LIN {X 0,Y 484.481,Z 413.449,A -85,B 0,C 180,E1 -6825.401,E2 -6825.401} C_VEL
LIN {X 0,Y 484,Z 426.052,A -85,B 0,C 180,E1 -6826.351,E2 -6826.351} C_VEL
LIN {X 0,Y 483.451,Z 437.461,A -85,B 0,C 180,E1 -6827.405,E2 -6827.405} C_VEL
LIN {X 0,Y 482.946,Z 446.93,A -85,B 0,C 180,E1 -6828.457,E2 -6828.457} C_VEL
LIN {X 0,Y 482.492,Z 456.426,A -85,B 0,C 180,E1 -6829.721,E2 -6829.721} C_VEL
LIN {X 0,Y 482.084,Z 465.497,A -85,B 0,C 180,E1 -6831.195,E2 -6831.195} C_VEL
LIN {X 0,Y 481.802,Z 471.841,A -85,B 0,C 180,E1 -6832.456,E2 -6832.456} C_VEL
LIN {X 0,Y 481.631,Z 477.067,A -85,B 0,C 180,E1 -6833.717,E2 -6833.717} C_VEL
LIN {X 0,Y 481.446,Z 482.599,A -85,B 0,C 180,E1 -6835.395,E2 -6835.395} C_VEL
LIN {X 0,Y 481.292,Z 485.698,A -85,B 0,C 180,E1 -6836.651,E2 -6836.651} C_VEL
LIN {X 0,Y 481.216,Z 488.621,A -85,B 0,C 180,E1 -6838.326,E2 -6838.326} C_VEL
LIN {X 0,Y 481.127,Z 490.218,A -85,B 0,C 180,E1 -6840,E2 -6840} C_VEL
LIN {X 0,Y 481.209,Z 490.492,A -85,B 0,C 180,E1 -6841.674,E2 -6841.674} C_VEL
LIN {X 0,Y 481.255,Z 489.477,A -85,B 0,C 180,E1 -6843.349,E2 -6843.349} C_VEL
LIN {X 0,Y 481.353,Z 487.122,A -85,B 0,C 180,E1 -6845.026,E2 -6845.026} C_VEL
LIN {X 0,Y 481.497,Z 484.405,A -85,B 0,C 180,E1 -6846.285,E2 -6846.285} C_VEL
LIN {X 0,Y 481.752,Z 479.514,A -85,B 0,C 180,E1 -6847.966,E2 -6847.966} C_VEL
LIN {X 0,Y 481.884,Z 474.735,A -85,B 0,C 180,E1 -6849.232,E2 -6849.232} C_VEL
LIN {X 0,Y 482.239,Z 467.834,A -85,B 0,C 180,E1 -6850.708,E2 -6850.708} C_VEL
LIN {X 0,Y 482.693,Z 459.289,A -85,B 0,C 180,E1 -6852.178,E2 -6852.178} C_VEL
LIN {X 0,Y 483.198,Z 450.109,A -85,B 0,C 180,E1 -6853.457,E2 -6853.457} C_VEL
LIN {X 0,Y 483.682,Z 438.95,A -85,B 0,C 180,E1 -6854.731,E2 -6854.731} C_VEL
LIN {X 0,Y 484.26,Z 427.523,A -85,B 0,C 180,E1 -6855.79,E2 -6855.79} C_VEL
LIN {X 0,Y 484.738,Z 415.459,A -85,B 0,C 180,E1 -6856.702,E2 -6856.702} C_VEL
LIN {X 0,Y 485.245,Z 402.361,A -85,B 0,C 180,E1 -6857.489,E2 -6857.489} C_VEL
LIN {X 0,Y 485.233,Z 400.246,A -85,B 0,C 180,E1 -6857.598,E2 -6857.598} C_VEL
LIN {X 0,Y 481.758,Z 389.103,A -85,B 0,C 180,E1 -6858.288,E2 -6858.288} C_VEL
LIN {X 0,Y 481.651,Z 389.119,A -85,B 0,C 180,E1 -6861.394,E2 -6861.394} C_VEL
LIN {X 0,Y 481.681,Z 389.115,A -85,B 0,C 180,E1 -6864.113,E2 -6864.113} C_VEL
LIN {X 0,Y 481.75,Z 389.103,A -85,B 0,C 180,E1 -6867.139,E2 -6867.139} C_VEL
LIN {X 0,Y 481.682,Z 389.111,A -85,B 0,C 180,E1 -6869.741,E2 -6869.741} C_VEL
LIN {X 0,Y 481.675,Z 389.113,A -85,B 0,C 180,E1 -6872.674,E2 -6872.674} C_VEL
LIN {X 0,Y 481.639,Z 389.117,A -85,B 0,C 180,E1 -6875.709,E2 -6875.709} C_VEL
LIN {X 0,Y 481.673,Z 389.114,A -85,B 0,C 180,E1 -6878.859,E2 -6878.859} C_VEL
LIN {X 0,Y 481.656,Z 389.115,A -85,B 0,C 180,E1 -6881.913,E2 -6881.913} C_VEL
LIN {X 0,Y 481.663,Z 389.116,A -85,B 0,C 180,E1 -6884.457,E2 -6884.457} C_VEL
LIN {X 0,Y 481.651,Z 389.119,A -85,B 0,C 180,E1 -6887.839,E2 -6887.839} C_VEL
LIN {X 0,Y 481.704,Z 389.203,A -85,B 0,C 180,E1 -6888.406,E2 -6888.406} C_VEL
LIN {X 0,Y 483.139,Z 396.916,A -85,B 0,C 180,E1 -6890.887,E2 -6890.887} C_VEL
LIN {X 0,Y 483.245,Z 401.045,A -85,B 0,C 180,E1 -6892.046,E2 -6892.046} C_VEL
LIN {X 0,Y 482.441,Z 414.228,A -85,B 0,C 180,E1 -6895.379,E2 -6895.379} C_VEL
LIN {X 0,Y 482.294,Z 426.909,A -85,B 0,C 180,E1 -6898.358,E2 -6898.358} C_VEL
LIN {X 0,Y 482.22,Z 439.845,A -85,B 0,C 180,E1 -6901.252,E2 -6901.252} C_VEL
LIN {X 0,Y 482.05,Z 455.738,A -85,B 0,C 180,E1 -6904.679,E2 -6904.679} C_VEL
LIN {X 0,Y 481.88,Z 471.239,A -85,B 0,C 180,E1 -6907.941,E2 -6907.941} C_VEL
LIN {X 0,Y 481.707,Z 486.219,A -85,B 0,C 180,E1 -6911.057,E2 -6911.057} C_VEL
LIN {X 0,Y 481.693,Z 490.574,A -85,B 0,C 180,E1 -6911.957,E2 -6911.957} C_VEL
LIN {X 0,Y 483.326,Z 507.533,A -85,B 0,C 180,E1 -6912.397,E2 -6912.397} C_VEL
LIN {X 0,Y 484.795,Z 517.449,A -85,B 0,C 180,E1 -6912.765,E2 -6912.765} C_VEL
LIN {X 0,Y 484.293,Z 531.486,A -85,B 0,C 180,E1 -6913.342,E2 -6913.342} C_VEL
LIN {X 0,Y 483.695,Z 545.297,A -85,B 0,C 180,E1 -6914.082,E2 -6914.082} C_VEL
LIN {X 0,Y 483.143,Z 559.303,A -85,B 0,C 180,E1 -6915.036,E2 -6915.036} C_VEL
LIN {X 0,Y 482.585,Z 571.818,A -85,B 0,C 180,E1 -6916.095,E2 -6916.095} C_VEL
LIN {X 0,Y 482.176,Z 582.238,A -85,B 0,C 180,E1 -6917.156,E2 -6917.156} C_VEL
LIN {X 0,Y 481.863,Z 592.671,A -85,B 0,C 180,E1 -6918.43,E2 -6918.43} C_VEL
LIN {X 0,Y 481.477,Z 601.314,A -85,B 0,C 180,E1 -6919.699,E2 -6919.699} C_VEL
LIN {X 0,Y 481.308,Z 609.635,A -85,B 0,C 180,E1 -6921.18,E2 -6921.18} C_VEL
LIN {X 0,Y 481.142,Z 615.438,A -85,B 0,C 180,E1 -6922.445,E2 -6922.445} C_VEL
LIN {X 0,Y 481.117,Z 620.135,A -85,B 0,C 180,E1 -6923.675,E2 -6923.675} C_VEL
LIN {X 0,Y 481.094,Z 624.005,A -85,B 0,C 180,E1 -6924.971,E2 -6924.971} C_VEL
LIN {X 0,Y 481.1,Z 626.043,A -85,B 0,C 180,E1 -6925.81,E2 -6925.81} C_VEL
LIN {X 0,Y 481.01,Z 628.967,A -85,B 0,C 180,E1 -6927.487,E2 -6927.487} C_VEL
LIN {X 0,Y 480.936,Z 630.44,A -85,B 0,C 180,E1 -6929.162,E2 -6929.162} C_VEL
LIN {X 0,Y 480.995,Z 630.658,A -85,B 0,C 180,E1 -6929.999,E2 -6929.999} C_VEL
LIN {X 0,Y 480.955,Z 630.008,A -85,B 0,C 180,E1 -6931.674,E2 -6931.674} C_VEL
LIN {X 0,Y 481.003,Z 627.954,A -85,B 0,C 180,E1 -6933.35,E2 -6933.35} C_VEL
LIN {X 0,Y 481.054,Z 624.44,A -85,B 0,C 180,E1 -6935.028,E2 -6935.028} C_VEL
LIN {X 0,Y 481.076,Z 619.364,A -85,B 0,C 180,E1 -6936.711,E2 -6936.711} C_VEL
LIN {X 0,Y 481.208,Z 612.595,A -85,B 0,C 180,E1 -6938.397,E2 -6938.397} C_VEL
LIN {X 0,Y 481.392,Z 605.054,A -85,B 0,C 180,E1 -6939.876,E2 -6939.876} C_VEL
LIN {X 0,Y 481.762,Z 595.692,A -85,B 0,C 180,E1 -6941.357,E2 -6941.357} C_VEL
LIN {X 0,Y 482.122,Z 585.91,A -85,B 0,C 180,E1 -6942.629,E2 -6942.629} C_VEL
LIN {X 0,Y 482.589,Z 575.113,A -85,B 0,C 180,E1 -6943.795,E2 -6943.795} C_VEL
LIN {X 0,Y 483.117,Z 563.234,A -85,B 0,C 180,E1 -6944.855,E2 -6944.855} C_VEL
LIN {X 0,Y 483.718,Z 551.697,A -85,B 0,C 180,E1 -6945.699,E2 -6945.699} C_VEL
LIN {X 0,Y 484.311,Z 539,A -85,B 0,C 180,E1 -6946.453,E2 -6946.453} C_VEL
LIN {X 0,Y 484.793,Z 525.706,A -85,B 0,C 180,E1 -6947.07,E2 -6947.07} C_VEL
LIN {X 0,Y 484.895,Z 515.976,A -85,B 0,C 180,E1 -6947.427,E2 -6947.427} C_VEL
LIN {X 0,Y 483.035,Z 503.611,A -85,B 0,C 180,E1 -6947.833,E2 -6947.833} C_VEL
LIN {X 0,Y 481.739,Z 494.305,A -85,B 0,C 180,E1 -6948.071,E2 -6948.071} C_VEL
LIN {X 0,Y 482.024,Z 480.891,A -85,B 0,C 180,E1 -6951.072,E2 -6951.072} C_VEL
LIN {X 0,Y 482.329,Z 469.472,A -85,B 0,C 180,E1 -6953.674,E2 -6953.674} C_VEL
LIN {X 0,Y 482.755,Z 455.849,A -85,B 0,C 180,E1 -6956.826,E2 -6956.826} C_VEL
LIN {X 0,Y 483.3,Z 442.011,A -85,B 0,C 180,E1 -6960.11,E2 -6960.11} C_VEL
LIN {X 0,Y 483.812,Z 428.138,A -85,B 0,C 180,E1 -6963.503,E2 -6963.503} C_VEL
LIN {X 0,Y 484.574,Z 413.921,A -85,B 0,C 180,E1 -6967.09,E2 -6967.09} C_VEL
LIN {X 0,Y 484.908,Z 406.263,A -85,B 0,C 180,E1 -6969.083,E2 -6969.083} C_VEL
LIN {X 0,Y 484.024,Z 400.159,A -85,B 0,C 180,E1 -6970.796,E2 -6970.796} C_VEL
LIN {X 0,Y 481.859,Z 390.061,A -85,B 0,C 180,E1 -6973.787,E2 -6973.787} C_VEL
LIN {X 0,Y 481.67,Z 389.114,A -85,B 0,C 180,E1 -6974.107,E2 -6974.107} C_VEL
LIN {X 0,Y 481.682,Z 389.107,A -85,B 0,C 180,E1 -6976.845,E2 -6976.845} C_VEL
LIN {X 0,Y 481.705,Z 389.108,A -85,B 0,C 180,E1 -6980.062,E2 -6980.062} C_VEL
LIN {X 0,Y 481.624,Z 389.118,A -85,B 0,C 180,E1 -6983.374,E2 -6983.374} C_VEL
LIN {X 0,Y 481.7,Z 389.106,A -85,B 0,C 180,E1 -6986.329,E2 -6986.329} C_VEL
LIN {X 0,Y 481.649,Z 389.116,A -85,B 0,C 180,E1 -6989.415,E2 -6989.415} C_VEL
LIN {X 0,Y 481.693,Z 389.108,A -85,B 0,C 180,E1 -6992.168,E2 -6992.168} C_VEL
LIN {X 0,Y 481.708,Z 389.105,A -85,B 0,C 180,E1 -6994.969,E2 -6994.969} C_VEL
LIN {X 0,Y 481.64,Z 389.115,A -85,B 0,C 180,E1 -6997.704,E2 -6997.704} C_VEL
LIN {X 0,Y 481.697,Z 389.106,A -85,B 0,C 180,E1 -7000.393,E2 -7000.393} C_VEL
LIN {X 0,Y 481.682,Z 389.109,A -85,B 0,C 180,E1 -7003.034,E2 -7003.034} C_VEL
LIN {X 0,Y 481.683,Z 389.11,A -85,B 0,C 180,E1 -7005.639,E2 -7005.639} C_VEL
LIN {X 0,Y 481.784,Z 389.096,A -85,B 0,C 180,E1 -7008.216,E2 -7008.216} C_VEL
LIN {X 0,Y 481.753,Z 389.101,A -85,B 0,C 180,E1 -7011.612,E2 -7011.612} C_VEL
LIN {X 0,Y 481.807,Z 389.093,A -85,B 0,C 180,E1 -7014.14,E2 -7014.14} C_VEL
LIN {X 0,Y 481.919,Z 389.081,A -85,B 0,C 180,E1 -7017.493,E2 -7017.493} C_VEL
LIN {X 0,Y 481.93,Z 389.078,A -85,B 0,C 180,E1 -7020,E2 -7020} C_VEL
LIN {X 0,Y 481.919,Z 389.078,A -85,B 0,C 180,E1 -7022.508,E2 -7022.508} C_VEL
LIN {X 0,Y 481.812,Z 389.093,A -85,B 0,C 180,E1 -7025.861,E2 -7025.861} C_VEL
LIN {X 0,Y 481.754,Z 389.099,A -85,B 0,C 180,E1 -7028.389,E2 -7028.389} C_VEL
LIN {X 0,Y 481.786,Z 389.096,A -85,B 0,C 180,E1 -7031.784,E2 -7031.784} C_VEL
LIN {X 0,Y 481.732,Z 389.105,A -85,B 0,C 180,E1 -7035.225,E2 -7035.225} C_VEL
LIN {X 0,Y 481.703,Z 389.106,A -85,B 0,C 180,E1 -7038.722,E2 -7038.722} C_VEL
LIN {X 0,Y 481.637,Z 389.116,A -85,B 0,C 180,E1 -7041.395,E2 -7041.395} C_VEL
LIN {X 0,Y 481.668,Z 389.11,A -85,B 0,C 180,E1 -7044.114,E2 -7044.114} C_VEL
LIN {X 0,Y 481.744,Z 389.104,A -85,B 0,C 180,E1 -7047.141,E2 -7047.141} C_VEL
LIN {X 0,Y 481.671,Z 389.111,A -85,B 0,C 180,E1 -7049.742,E2 -7049.742} C_VEL
LIN {X 0,Y 481.666,Z 389.111,A -85,B 0,C 180,E1 -7052.675,E2 -7052.675} C_VEL
LIN {X 0,Y 481.636,Z 389.115,A -85,B 0,C 180,E1 -7055.71,E2 -7055.71} C_VEL
LIN {X 0,Y 481.665,Z 389.114,A -85,B 0,C 180,E1 -7058.86,E2 -7058.86} C_VEL
LIN {X 0,Y 481.657,Z 389.111,A -85,B 0,C 180,E1 -7061.915,E2 -7061.915} C_VEL
LIN {X 0,Y 481.655,Z 389.112,A -85,B 0,C 180,E1 -7064.458,E2 -7064.458} C_VEL
LIN {X 0,Y 481.645,Z 389.113,A -85,B 0,C 180,E1 -7067.841,E2 -7067.841} C_VEL
LIN {X 0,Y 481.716,Z 389.106,A -85,B 0,C 180,E1 -7070.647,E2 -7070.647} C_VEL
LIN {X 0,Y 481.641,Z 389.113,A -85,B 0,C 180,E1 -7074.292,E2 -7074.292} C_VEL
LIN {X 0,Y 481.672,Z 389.111,A -85,B 0,C 180,E1 -7077.327,E2 -7077.327} C_VEL
LIN {X 0,Y 481.678,Z 389.109,A -85,B 0,C 180,E1 -7080.26,E2 -7080.26} C_VEL
LIN {X 0,Y 481.745,Z 389.102,A -85,B 0,C 180,E1 -7083.113,E2 -7083.113} C_VEL
LIN {X 0,Y 481.674,Z 389.109,A -85,B 0,C 180,E1 -7085.888,E2 -7085.888} C_VEL
LIN {X 0,Y 481.636,Z 389.113,A -85,B 0,C 180,E1 -7087.993,E2 -7087.993} C_VEL
LIN {X 0,Y 480.97,Z 389.201,A -85,B 0,C 180,E1 -7088.691,E2 -7088.691} C_VEL
LIN {X 0,Y 478.144,Z 389.55,A -85,B 0,C 180,E1 -7089.826,E2 -7089.826} C_VEL
LIN {X 0,Y 475.759,Z 389.85,A -85,B 0,C 180,E1 -7090.74,E2 -7090.74} C_VEL
LIN {X 0,Y 474.738,Z 389.974,A -85,B 0,C 180,E1 -7091.446,E2 -7091.446} C_VEL
LIN {X 0,Y 474.656,Z 389.983,A -85,B 0,C 180,E1 -7091.685,E2 -7091.685} C_VEL
LIN {X 0,Y 474.667,Z 389.985,A -85,B 0,C 180,E1 -7094.544,E2 -7094.544} C_VEL
LIN {X 0,Y 474.411,Z 390.02,A -85,B 0,C 180,E1 -7097.971,E2 -7097.971} C_VEL
LIN {X 0,Y 477.563,Z 400.909,A -85,B 0,C 180,E1 -7098.38,E2 -7098.38} C_VEL
LIN {X 0,Y 477.396,Z 412.945,A -85,B 0,C 180,E1 -7098.86,E2 -7098.86} C_VEL
LIN {X 0,Y 477.088,Z 424.636,A -85,B 0,C 180,E1 -7099.498,E2 -7099.498} C_VEL
LIN {X 0,Y 476.667,Z 436.587,A -85,B 0,C 180,E1 -7100.346,E2 -7100.346} C_VEL
LIN {X 0,Y 476.218,Z 447.382,A -85,B 0,C 180,E1 -7101.322,E2 -7101.322} C_VEL
LIN {X 0,Y 475.777,Z 456.619,A -85,B 0,C 180,E1 -7102.361,E2 -7102.361} C_VEL
LIN {X 0,Y 475.463,Z 465.754,A -85,B 0,C 180,E1 -7103.636,E2 -7103.636} C_VEL
LIN {X 0,Y 475.01,Z 473.056,A -85,B 0,C 180,E1 -7104.908,E2 -7104.908} C_VEL
LIN {X 0,Y 474.819,Z 478.896,A -85,B 0,C 180,E1 -7106.182,E2 -7106.182} C_VEL
LIN {X 0,Y 474.549,Z 483.539,A -85,B 0,C 180,E1 -7107.454,E2 -7107.454} C_VEL
LIN {X 0,Y 474.42,Z 487.086,A -85,B 0,C 180,E1 -7108.728,E2 -7108.728} C_VEL
LIN {X 0,Y 474.264,Z 489.665,A -85,B 0,C 180,E1 -7110.001,E2 -7110.001} C_VEL
LIN {X 0,Y 474.172,Z 490.883,A -85,B 0,C 180,E1 -7110.85,E2 -7110.85} C_VEL
LIN {X 0,Y 474.231,Z 491.699,A -85,B 0,C 180,E1 -7111.699,E2 -7111.699} C_VEL
LIN {X 0,Y 474.199,Z 492.137,A -85,B 0,C 180,E1 -7113.4,E2 -7113.4} C_VEL
LIN {X 0,Y 474.326,Z 491.062,A -85,B 0,C 180,E1 -7115.101,E2 -7115.101} C_VEL
LIN {X 0,Y 474.401,Z 488.37,A -85,B 0,C 180,E1 -7116.807,E2 -7116.807} C_VEL
LIN {X 0,Y 474.51,Z 485.252,A -85,B 0,C 180,E1 -7118.089,E2 -7118.089} C_VEL
LIN {X 0,Y 474.746,Z 481.073,A -85,B 0,C 180,E1 -7119.373,E2 -7119.373} C_VEL
LIN {X 0,Y 475,Z 475.726,A -85,B 0,C 180,E1 -7120.659,E2 -7120.659} C_VEL
LIN {X 0,Y 475.219,Z 469.012,A -85,B 0,C 180,E1 -7121.95,E2 -7121.95} C_VEL
LIN {X 0,Y 475.672,Z 460.54,A -85,B 0,C 180,E1 -7123.24,E2 -7123.24} C_VEL
LIN {X 0,Y 476.07,Z 451.844,A -85,B 0,C 180,E1 -7124.317,E2 -7124.317} C_VEL
LIN {X 0,Y 476.483,Z 442.254,A -85,B 0,C 180,E1 -7125.288,E2 -7125.288} C_VEL
LIN {X 0,Y 476.917,Z 431.6,A -85,B 0,C 180,E1 -7126.15,E2 -7126.15} C_VEL
LIN {X 0,Y 477.284,Z 419.943,A -85,B 0,C 180,E1 -7126.895,E2 -7126.895} C_VEL
LIN {X 0,Y 477.516,Z 408.575,A -85,B 0,C 180,E1 -7127.451,E2 -7127.451} C_VEL
LIN {X 0,Y 477.528,Z 400.444,A -85,B 0,C 180,E1 -7127.755,E2 -7127.755} C_VEL
LIN {X 0,Y 474.357,Z 390.025,A -85,B 0,C 180,E1 -7128.162,E2 -7128.162} C_VEL
LIN {X 0,Y 474.575,Z 389.998,A -85,B 0,C 180,E1 -7131.096,E2 -7131.096} C_VEL
LIN {X 0,Y 474.663,Z 389.982,A -85,B 0,C 180,E1 -7134.493,E2 -7134.493} C_VEL
LIN {X 0,Y 474.687,Z 389.981,A -85,B 0,C 180,E1 -7137.335,E2 -7137.335} C_VEL
LIN {X 0,Y 474.611,Z 389.99,A -85,B 0,C 180,E1 -7140.23,E2 -7140.23} C_VEL
LIN {X 0,Y 474.631,Z 389.989,A -85,B 0,C 180,E1 -7143.222,E2 -7143.222} C_VEL
LIN {X 0,Y 474.594,Z 389.994,A -85,B 0,C 180,E1 -7146.324,E2 -7146.324} C_VEL
LIN {X 0,Y 474.623,Z 389.983,A -85,B 0,C 180,E1 -7149.646,E2 -7149.646} C_VEL
LIN {X 0,Y 474.62,Z 389.988,A -85,B 0,C 180,E1 -7152.934,E2 -7152.934} C_VEL
LIN {X 0,Y 474.621,Z 389.986,A -85,B 0,C 180,E1 -7155.896,E2 -7155.896} C_VEL
LIN {X 0,Y 474.638,Z 389.98,A -85,B 0,C 180,E1 -7159.04,E2 -7159.04} C_VEL
LIN {X 0,Y 474.616,Z 389.973,A -85,B 0,C 180,E1 -7161.704,E2 -7161.704} C_VEL
LIN {X 0,Y 474.634,Z 389.985,A -85,B 0,C 180,E1 -7164.726,E2 -7164.726} C_VEL
LIN {X 0,Y 474.64,Z 389.984,A -85,B 0,C 180,E1 -7167.788,E2 -7167.788} C_VEL
LIN {X 0,Y 474.627,Z 389.966,A -85,B 0,C 180,E1 -7170.885,E2 -7170.885} C_VEL
LIN {X 0,Y 474.658,Z 389.981,A -85,B 0,C 180,E1 -7173.628,E2 -7173.628} C_VEL
LIN {X 0,Y 474.639,Z 389.984,A -85,B 0,C 180,E1 -7176.642,E2 -7176.642} C_VEL
LIN {X 0,Y 474.658,Z 389.983,A -85,B 0,C 180,E1 -7180.089,E2 -7180.089} C_VEL
LIN {X 0,Y 474.643,Z 389.986,A -85,B 0,C 180,E1 -7182.774,E2 -7182.774} C_VEL
LIN {X 0,Y 474.66,Z 389.987,A -85,B 0,C 180,E1 -7183.698,E2 -7183.698} C_VEL
LIN {X 0,Y 478.112,Z 401.182,A -85,B 0,C 180,E1 -7184.391,E2 -7184.391} C_VEL
LIN {X 0,Y 477.676,Z 414.246,A -85,B 0,C 180,E1 -7185.188,E2 -7185.188} C_VEL
LIN {X 0,Y 477.171,Z 426.871,A -85,B 0,C 180,E1 -7186.152,E2 -7186.152} C_VEL
LIN {X 0,Y 476.591,Z 438.305,A -85,B 0,C 180,E1 -7187.22,E2 -7187.22} C_VEL
LIN {X 0,Y 476.047,Z 447.801,A -85,B 0,C 180,E1 -7188.288,E2 -7188.288} C_VEL
LIN {X 0,Y 475.566,Z 457.324,A -85,B 0,C 180,E1 -7189.57,E2 -7189.57} C_VEL
LIN {X 0,Y 475.14,Z 466.422,A -85,B 0,C 180,E1 -7191.065,E2 -7191.065} C_VEL
LIN {X 0,Y 474.77,Z 474.16,A -85,B 0,C 180,E1 -7192.659,E2 -7192.659} C_VEL
LIN {X 0,Y 474.568,Z 479.586,A -85,B 0,C 180,E1 -7194.05,E2 -7194.05} C_VEL
LIN {X 0,Y 474.371,Z 484.706,A -85,B 0,C 180,E1 -7195.752,E2 -7195.752} C_VEL
LIN {X 0,Y 474.191,Z 488.351,A -85,B 0,C 180,E1 -7197.451,E2 -7197.451} C_VEL
LIN {X 0,Y 474.131,Z 490.614,A -85,B 0,C 180,E1 -7199.15,E2 -7199.15} C_VEL
LIN {X 0,Y 474.13,Z 491.557,A -85,B 0,C 180,E1 -7200.849,E2 -7200.849} C_VEL
LIN {X 0,Y 474.188,Z 491.196,A -85,B 0,C 180,E1 -7202.548,E2 -7202.548} C_VEL
LIN {X 0,Y 474.302,Z 489.516,A -85,B 0,C 180,E1 -7204.249,E2 -7204.249} C_VEL
LIN {X 0,Y 474.548,Z 486.437,A -85,B 0,C 180,E1 -7205.95,E2 -7205.95} C_VEL
LIN {X 0,Y 474.668,Z 481.914,A -85,B 0,C 180,E1 -7207.658,E2 -7207.658} C_VEL
LIN {X 0,Y 474.946,Z 475.768,A -85,B 0,C 180,E1 -7209.368,E2 -7209.368} C_VEL
LIN {X 0,Y 475.329,Z 468.849,A -85,B 0,C 180,E1 -7210.866,E2 -7210.866} C_VEL
LIN {X 0,Y 475.825,Z 460.26,A -85,B 0,C 180,E1 -7212.356,E2 -7212.356} C_VEL
LIN {X 0,Y 476.362,Z 451.042,A -85,B 0,C 180,E1 -7213.654,E2 -7213.654} C_VEL
LIN {X 0,Y 476.897,Z 439.881,A -85,B 0,C 180,E1 -7214.945,E2 -7214.945} C_VEL
LIN {X 0,Y 477.509,Z 428.474,A -85,B 0,C 180,E1 -7216.019,E2 -7216.019} C_VEL
LIN {X 0,Y 478.025,Z 416.614,A -85,B 0,C 180,E1 -7216.931,E2 -7216.931} C_VEL
LIN {X 0,Y 478.544,Z 403.318,A -85,B 0,C 180,E1 -7217.742,E2 -7217.742} C_VEL
LIN {X 0,Y 478.234,Z 401.241,A -85,B 0,C 180,E1 -7217.865,E2 -7217.865} C_VEL
LIN {X 0,Y 474.681,Z 389.984,A -85,B 0,C 180,E1 -7218.584,E2 -7218.584} C_VEL
LIN {X 0,Y 474.638,Z 389.99,A -85,B 0,C 180,E1 -7221.116,E2 -7221.116} C_VEL
LIN {X 0,Y 474.662,Z 389.988,A -85,B 0,C 180,E1 -7224.493,E2 -7224.493} C_VEL
LIN {X 0,Y 474.684,Z 389.983,A -85,B 0,C 180,E1 -7227.334,E2 -7227.334} C_VEL
LIN {X 0,Y 474.608,Z 389.992,A -85,B 0,C 180,E1 -7230.23,E2 -7230.23} C_VEL
LIN {X 0,Y 474.646,Z 389.987,A -85,B 0,C 180,E1 -7233.22,E2 -7233.22} C_VEL
LIN {X 0,Y 474.591,Z 389.995,A -85,B 0,C 180,E1 -7236.323,E2 -7236.323} C_VEL
LIN {X 0,Y 474.63,Z 389.99,A -85,B 0,C 180,E1 -7239.647,E2 -7239.647} C_VEL
LIN {X 0,Y 474.618,Z 389.993,A -85,B 0,C 180,E1 -7242.934,E2 -7242.934} C_VEL
LIN {X 0,Y 474.612,Z 389.995,A -85,B 0,C 180,E1 -7245.895,E2 -7245.895} C_VEL
LIN {X 0,Y 474.65,Z 390.163,A -85,B 0,C 180,E1 -7248.052,E2 -7248.052} C_VEL
LIN {X 0,Y 476.134,Z 397.733,A -85,B 0,C 180,E1 -7250.601,E2 -7250.601} C_VEL
LIN {X 0,Y 476.361,Z 401.493,A -85,B 0,C 180,E1 -7251.709,E2 -7251.709} C_VEL
LIN {X 0,Y 475.557,Z 413.309,A -85,B 0,C 180,E1 -7254.804,E2 -7254.804} C_VEL
LIN {X 0,Y 475.279,Z 426.858,A -85,B 0,C 180,E1 -7258.086,E2 -7258.086} C_VEL
LIN {X 0,Y 475.182,Z 439.702,A -85,B 0,C 180,E1 -7261.028,E2 -7261.028} C_VEL
LIN {X 0,Y 474.98,Z 455.881,A -85,B 0,C 180,E1 -7264.589,E2 -7264.589} C_VEL
LIN {X 0,Y 474.799,Z 469.882,A -85,B 0,C 180,E1 -7267.594,E2 -7267.594} C_VEL
LIN {X 0,Y 474.667,Z 484.848,A -85,B 0,C 180,E1 -7270.765,E2 -7270.765} C_VEL
LIN {X 0,Y 474.625,Z 489.143,A -85,B 0,C 180,E1 -7271.671,E2 -7271.671} C_VEL
LIN {X 0,Y 476.247,Z 506.063,A -85,B 0,C 180,E1 -7272.127,E2 -7272.127} C_VEL
LIN {X 0,Y 477.39,Z 514.673,A -85,B 0,C 180,E1 -7272.448,E2 -7272.448} C_VEL
LIN {X 0,Y 477.842,Z 518.839,A -85,B 0,C 180,E1 -7272.617,E2 -7272.617} C_VEL
LIN {X 0,Y 477.327,Z 531.995,A -85,B 0,C 180,E1 -7273.194,E2 -7273.194} C_VEL
LIN {X 0,Y 476.708,Z 545.487,A -85,B 0,C 180,E1 -7273.952,E2 -7273.952} C_VEL
LIN {X 0,Y 476.112,Z 559.127,A -85,B 0,C 180,E1 -7274.919,E2 -7274.919} C_VEL
LIN {X 0,Y 475.54,Z 571.477,A -85,B 0,C 180,E1 -7275.994,E2 -7275.994} C_VEL
LIN {X 0,Y 475.069,Z 582.717,A -85,B 0,C 180,E1 -7277.178,E2 -7277.178} C_VEL
LIN {X 0,Y 474.747,Z 592.909,A -85,B 0,C 180,E1 -7278.471,E2 -7278.471} C_VEL
LIN {X 0,Y 474.373,Z 601.353,A -85,B 0,C 180,E1 -7279.758,E2 -7279.758} C_VEL
LIN {X 0,Y 474.231,Z 608.412,A -85,B 0,C 180,E1 -7281.047,E2 -7281.047} C_VEL
LIN {X 0,Y 474.088,Z 614.264,A -85,B 0,C 180,E1 -7282.332,E2 -7282.332} C_VEL
LIN {X 0,Y 474.072,Z 619.213,A -85,B 0,C 180,E1 -7283.647,E2 -7283.647} C_VEL
LIN {X 0,Y 474.045,Z 623.981,A -85,B 0,C 180,E1 -7285.322,E2 -7285.322} C_VEL
LIN {X 0,Y 474.002,Z 626.623,A -85,B 0,C 180,E1 -7286.599,E2 -7286.599} C_VEL
LIN {X 0,Y 473.943,Z 628.848,A -85,B 0,C 180,E1 -7288.3,E2 -7288.3} C_VEL
LIN {X 0,Y 473.986,Z 629.648,A -85,B 0,C 180,E1 -7289.999,E2 -7289.999} C_VEL
LIN {X 0,Y 473.921,Z 629.009,A -85,B 0,C 180,E1 -7291.699,E2 -7291.699} C_VEL
LIN {X 0,Y 473.96,Z 626.961,A -85,B 0,C 180,E1 -7293.399,E2 -7293.399} C_VEL
LIN {X 0,Y 474.003,Z 623.448,A -85,B 0,C 180,E1 -7295.103,E2 -7295.103} C_VEL
LIN {X 0,Y 474.01,Z 618.372,A -85,B 0,C 180,E1 -7296.811,E2 -7296.811} C_VEL
LIN {X 0,Y 474.129,Z 611.594,A -85,B 0,C 180,E1 -7298.523,E2 -7298.523} C_VEL
LIN {X 0,Y 474.331,Z 604.042,A -85,B 0,C 180,E1 -7300.025,E2 -7300.025} C_VEL
LIN {X 0,Y 474.738,Z 594.663,A -85,B 0,C 180,E1 -7301.527,E2 -7301.527} C_VEL
LIN {X 0,Y 475.103,Z 584.867,A -85,B 0,C 180,E1 -7302.819,E2 -7302.819} C_VEL
LIN {X 0,Y 475.571,Z 574.055,A -85,B 0,C 180,E1 -7304.003,E2 -7304.003} C_VEL
LIN {X 0,Y 476.175,Z 562.167,A -85,B 0,C 180,E1 -7305.077,E2 -7305.077} C_VEL
LIN {X 0,Y 476.906,Z 549.046,A -85,B 0,C 180,E1 -7306.039,E2 -7306.039} C_VEL
LIN {X 0,Y 477.519,Z 535.992,A -85,B 0,C 180,E1 -7306.801,E2 -7306.801} C_VEL
LIN {X 0,Y 477.984,Z 523.331,A -85,B 0,C 180,E1 -7307.376,E2 -7307.376} C_VEL
LIN {X 0,Y 478.046,Z 517.123,A -85,B 0,C 180,E1 -7307.608,E2 -7307.608} C_VEL
LIN {X 0,Y 476.051,Z 503.386,A -85,B 0,C 180,E1 -7308.08,E2 -7308.08} C_VEL
LIN {X 0,Y 474.688,Z 493.54,A -85,B 0,C 180,E1 -7308.336,E2 -7308.336} C_VEL
LIN {X 0,Y 475.01,Z 480.065,A -85,B 0,C 180,E1 -7311.415,E2 -7311.415} C_VEL
LIN {X 0,Y 475.38,Z 466.973,A -85,B 0,C 180,E1 -7314.452,E2 -7314.452} C_VEL
LIN {X 0,Y 475.796,Z 455.143,A -85,B 0,C 180,E1 -7317.25,E2 -7317.25} C_VEL
LIN {X 0,Y 476.351,Z 441.309,A -85,B 0,C 180,E1 -7320.596,E2 -7320.596} C_VEL
LIN {X 0,Y 476.849,Z 429.407,A -85,B 0,C 180,E1 -7323.55,E2 -7323.55} C_VEL
LIN {X 0,Y 477.678,Z 414.426,A -85,B 0,C 180,E1 -7327.393,E2 -7327.393} C_VEL
LIN {X 0,Y 478.018,Z 407.568,A -85,B 0,C 180,E1 -7329.211,E2 -7329.211} C_VEL
LIN {X 0,Y 477.157,Z 401.904,A -85,B 0,C 180,E1 -7330.818,E2 -7330.818} C_VEL
LIN {X 0,Y 475.177,Z 392.768,A -85,B 0,C 180,E1 -7333.554,E2 -7333.554} C_VEL
LIN {X 0,Y 474.613,Z 389.992,A -85,B 0,C 180,E1 -7334.456,E2 -7334.456} C_VEL
LIN {X 0,Y 474.643,Z 389.989,A -85,B 0,C 180,E1 -7337.759,E2 -7337.759} C_VEL
LIN {X 0,Y 474.674,Z 389.981,A -85,B 0,C 180,E1 -7340.457,E2 -7340.457} C_VEL
LIN {X 0,Y 474.585,Z 389.995,A -85,B 0,C 180,E1 -7343.676,E2 -7343.676} C_VEL
LIN {X 0,Y 474.634,Z 389.986,A -85,B 0,C 180,E1 -7346.779,E2 -7346.779} C_VEL
LIN {X 0,Y 474.604,Z 389.992,A -85,B 0,C 180,E1 -7349.77,E2 -7349.77} C_VEL
LIN {X 0,Y 474.704,Z 389.977,A -85,B 0,C 180,E1 -7352.68,E2 -7352.68} C_VEL
LIN {X 0,Y 474.649,Z 389.988,A -85,B 0,C 180,E1 -7355.507,E2 -7355.507} C_VEL
LIN {X 0,Y 474.66,Z 389.985,A -85,B 0,C 180,E1 -7359.185,E2 -7359.185} C_VEL
LIN {X 0,Y 474.646,Z 389.985,A -85,B 0,C 180,E1 -7361.884,E2 -7361.884} C_VEL
LIN {X 0,Y 474.69,Z 389.979,A -85,B 0,C 180,E1 -7364.544,E2 -7364.544} C_VEL
LIN {X 0,Y 474.728,Z 389.975,A -85,B 0,C 180,E1 -7368.038,E2 -7368.038} C_VEL
LIN {X 0,Y 474.718,Z 389.978,A -85,B 0,C 180,E1 -7371.486,E2 -7371.486} C_VEL
LIN {X 0,Y 474.769,Z 389.97,A -85,B 0,C 180,E1 -7374.052,E2 -7374.052} C_VEL
LIN {X 0,Y 474.885,Z 389.957,A -85,B 0,C 180,E1 -7377.456,E2 -7377.456} C_VEL
LIN {X 0,Y 474.867,Z 389.958,A -85,B 0,C 180,E1 -7380.848,E2 -7380.848} C_VEL
LIN {X 0,Y 474.885,Z 389.954,A -85,B 0,C 180,E1 -7382.545,E2 -7382.545} C_VEL
LIN {X 0,Y 474.773,Z 389.97,A -85,B 0,C 180,E1 -7385.948,E2 -7385.948} C_VEL
LIN {X 0,Y 474.719,Z 389.975,A -85,B 0,C 180,E1 -7388.514,E2 -7388.514} C_VEL
LIN {X 0,Y 474.729,Z 389.975,A -85,B 0,C 180,E1 -7391.962,E2 -7391.962} C_VEL
LIN {X 0,Y 474.67,Z 389.982,A -85,B 0,C 180,E1 -7395.769,E2 -7395.769} C_VEL
LIN {X 0,Y 474.656,Z 389.987,A -85,B 0,C 180,E1 -7399.011,E2 -7399.011} C_VEL
LIN {X 0,Y 474.581,Z 389.993,A -85,B 0,C 180,E1 -7401.73,E2 -7401.73} C_VEL
LIN {X 0,Y 474.65,Z 389.984,A -85,B 0,C 180,E1 -7404.494,E2 -7404.494} C_VEL
LIN {X 0,Y 474.69,Z 389.981,A -85,B 0,C 180,E1 -7407.34,E2 -7407.34} C_VEL
LIN {X 0,Y 474.597,Z 389.993,A -85,B 0,C 180,E1 -7410.811,E2 -7410.811} C_VEL
LIN {X 0,Y 474.631,Z 389.987,A -85,B 0,C 180,E1 -7413.985,E2 -7413.985} C_VEL
LIN {X 0,Y 474.569,Z 389.998,A -85,B 0,C 180,E1 -7416.901,E2 -7416.901} C_VEL
LIN {X 0,Y 474.622,Z 389.989,A -85,B 0,C 180,E1 -7419.649,E2 -7419.649} C_VEL
LIN {X 0,Y 474.639,Z 389.99,A -85,B 0,C 180,E1 -7422.932,E2 -7422.932} C_VEL
LIN {X 0,Y 474.604,Z 389.99,A -85,B 0,C 180,E1 -7425.896,E2 -7425.896} C_VEL
LIN {X 0,Y 474.637,Z 389.988,A -85,B 0,C 180,E1 -7429.04,E2 -7429.04} C_VEL
LIN {X 0,Y 474.616,Z 389.989,A -85,B 0,C 180,E1 -7431.704,E2 -7431.704} C_VEL
LIN {X 0,Y 474.628,Z 389.99,A -85,B 0,C 180,E1 -7434.728,E2 -7434.728} C_VEL
LIN {X 0,Y 474.636,Z 389.986,A -85,B 0,C 180,E1 -7437.789,E2 -7437.789} C_VEL
LIN {X 0,Y 474.624,Z 389.991,A -85,B 0,C 180,E1 -7440.886,E2 -7440.886} C_VEL
LIN {X 0,Y 474.66,Z 389.984,A -85,B 0,C 180,E1 -7443.63,E2 -7443.63} C_VEL
LIN {X 0,Y 474.636,Z 389.989,A -85,B 0,C 180,E1 -7446.643,E2 -7446.643} C_VEL
LIN {X 0,Y 474.656,Z 389.983,A -85,B 0,C 180,E1 -7450.091,E2 -7450.091} C_VEL
LIN {X 0,Y 474.656,Z 389.983,A -85,B 0,C 180,E1 -7451.685,E2 -7451.685} C_VEL
LIN {X 0,Y 473.99,Z 390.069,A -85,B 0,C 180,E1 -7452.393,E2 -7452.393} C_VEL
LIN {X 0,Y 471.126,Z 390.425,A -85,B 0,C 180,E1 -7453.544,E2 -7453.544} C_VEL
LIN {X 0,Y 468.683,Z 390.73,A -85,B 0,C 180,E1 -7454.472,E2 -7454.472} C_VEL
LIN {X 0,Y 467.609,Z 390.864,A -85,B 0,C 180,E1 -7455.189,E2 -7455.189} C_VEL
LIN {X 0,Y 467.509,Z 390.876,A -85,B 0,C 180,E1 -7455.432,E2 -7455.432} C_VEL
LIN {X 0,Y 467.388,Z 390.895,A -85,B 0,C 180,E1 -7457.736,E2 -7457.736} C_VEL
LIN {X 0,Y 470.729,Z 402.115,A -85,B 0,C 180,E1 -7458.181,E2 -7458.181} C_VEL
LIN {X 0,Y 470.535,Z 414.749,A -85,B 0,C 180,E1 -7458.7,E2 -7458.7} C_VEL
LIN {X 0,Y 470.22,Z 426.175,A -85,B 0,C 180,E1 -7459.342,E2 -7459.342} C_VEL
LIN {X 0,Y 469.775,Z 438.031,A -85,B 0,C 180,E1 -7460.203,E2 -7460.203} C_VEL
LIN {X 0,Y 469.326,Z 448.715,A -85,B 0,C 180,E1 -7461.194,E2 -7461.194} C_VEL
LIN {X 0,Y 468.86,Z 457.9,A -85,B 0,C 180,E1 -7462.248,E2 -7462.248} C_VEL
LIN {X 0,Y 468.518,Z 466.982,A -85,B 0,C 180,E1 -7463.541,E2 -7463.541} C_VEL
LIN {X 0,Y 468.036,Z 474.24,A -85,B 0,C 180,E1 -7464.832,E2 -7464.832} C_VEL
LIN {X 0,Y 467.838,Z 480.046,A -85,B 0,C 180,E1 -7466.125,E2 -7466.125} C_VEL
LIN {X 0,Y 467.563,Z 484.657,A -85,B 0,C 180,E1 -7467.416,E2 -7467.416} C_VEL
LIN {X 0,Y 467.419,Z 488.176,A -85,B 0,C 180,E1 -7468.709,E2 -7468.709} C_VEL
LIN {X 0,Y 467.258,Z 490.727,A -85,B 0,C 180,E1 -7470.001,E2 -7470.001} C_VEL
LIN {X 0,Y 467.152,Z 491.933,A -85,B 0,C 180,E1 -7470.863,E2 -7470.863} C_VEL
LIN {X 0,Y 467.214,Z 492.726,A -85,B 0,C 180,E1 -7471.725,E2 -7471.725} C_VEL
LIN {X 0,Y 467.172,Z 493.135,A -85,B 0,C 180,E1 -7473.451,E2 -7473.451} C_VEL
LIN {X 0,Y 467.217,Z 492.779,A -85,B 0,C 180,E1 -7474.314,E2 -7474.314} C_VEL
LIN {X 0,Y 467.321,Z 492.018,A -85,B 0,C 180,E1 -7475.178,E2 -7475.178} C_VEL
LIN {X 0,Y 467.404,Z 489.299,A -85,B 0,C 180,E1 -7476.91,E2 -7476.91} C_VEL
LIN {X 0,Y 467.539,Z 486.15,A -85,B 0,C 180,E1 -7478.211,E2 -7478.211} C_VEL
LIN {X 0,Y 467.791,Z 481.94,A -85,B 0,C 180,E1 -7479.513,E2 -7479.513} C_VEL
LIN {X 0,Y 468.066,Z 476.559,A -85,B 0,C 180,E1 -7480.819,E2 -7480.819} C_VEL
LIN {X 0,Y 468.311,Z 469.79,A -85,B 0,C 180,E1 -7482.129,E2 -7482.129} C_VEL
LIN {X 0,Y 468.803,Z 461.271,A -85,B 0,C 180,E1 -7483.437,E2 -7483.437} C_VEL
LIN {X 0,Y 469.225,Z 452.523,A -85,B 0,C 180,E1 -7484.53,E2 -7484.53} C_VEL
LIN {X 0,Y 469.659,Z 442.835,A -85,B 0,C 180,E1 -7485.515,E2 -7485.515} C_VEL
LIN {X 0,Y 470.113,Z 432.085,A -85,B 0,C 180,E1 -7486.391,E2 -7486.391} C_VEL
LIN {X 0,Y 470.5,Z 420.71,A -85,B 0,C 180,E1 -7487.122,E2 -7487.122} C_VEL
LIN {X 0,Y 470.733,Z 408.667,A -85,B 0,C 180,E1 -7487.711,E2 -7487.711} C_VEL
LIN {X 0,Y 470.654,Z 401.548,A -85,B 0,C 180,E1 -7487.981,E2 -7487.981} C_VEL
LIN {X 0,Y 467.312,Z 390.903,A -85,B 0,C 180,E1 -7488.411,E2 -7488.411} C_VEL
LIN {X 0,Y 467.534,Z 390.875,A -85,B 0,C 180,E1 -7491.252,E2 -7491.252} C_VEL
LIN {X 0,Y 467.578,Z 390.863,A -85,B 0,C 180,E1 -7493.944,E2 -7493.944} C_VEL
LIN {X 0,Y 467.623,Z 390.863,A -85,B 0,C 180,E1 -7496.801,E2 -7496.801} C_VEL
LIN {X 0,Y 467.56,Z 390.867,A -85,B 0,C 180,E1 -7499.738,E2 -7499.738} C_VEL
LIN {X 0,Y 467.585,Z 390.869,A -85,B 0,C 180,E1 -7502.759,E2 -7502.759} C_VEL
LIN {X 0,Y 467.559,Z 390.868,A -85,B 0,C 180,E1 -7505.89,E2 -7505.89} C_VEL
LIN {X 0,Y 467.581,Z 390.862,A -85,B 0,C 180,E1 -7509.145,E2 -7509.145} C_VEL
LIN {X 0,Y 467.592,Z 390.866,A -85,B 0,C 180,E1 -7512.567,E2 -7512.567} C_VEL
LIN {X 0,Y 467.576,Z 390.862,A -85,B 0,C 180,E1 -7515.053,E2 -7515.053} C_VEL
LIN {X 0,Y 467.594,Z 390.861,A -85,B 0,C 180,E1 -7517.44,E2 -7517.44} C_VEL
LIN {X 0,Y 467.587,Z 390.847,A -85,B 0,C 180,E1 -7520.855,E2 -7520.855} C_VEL
LIN {X 0,Y 467.568,Z 390.87,A -85,B 0,C 180,E1 -7524.26,E2 -7524.26} C_VEL
LIN {X 0,Y 467.586,Z 390.861,A -85,B 0,C 180,E1 -7527.321,E2 -7527.321} C_VEL
LIN {X 0,Y 467.573,Z 390.845,A -85,B 0,C 180,E1 -7530.668,E2 -7530.668} C_VEL
LIN {X 0,Y 467.617,Z 390.853,A -85,B 0,C 180,E1 -7533.199,E2 -7533.199} C_VEL
LIN {X 0,Y 467.595,Z 390.862,A -85,B 0,C 180,E1 -7536.469,E2 -7536.469} C_VEL
LIN {X 0,Y 467.626,Z 390.862,A -85,B 0,C 180,E1 -7539.777,E2 -7539.777} C_VEL
LIN {X 0,Y 467.602,Z 390.862,A -85,B 0,C 180,E1 -7542.506,E2 -7542.506} C_VEL
LIN {X 0,Y 467.589,Z 390.869,A -85,B 0,C 180,E1 -7543.449,E2 -7543.449} C_VEL
LIN {X 0,Y 471.384,Z 403.663,A -85,B 0,C 180,E1 -7544.264,E2 -7544.264} C_VEL
LIN {X 0,Y 470.848,Z 416.539,A -85,B 0,C 180,E1 -7545.079,E2 -7545.079} C_VEL
LIN {X 0,Y 470.278,Z 428.914,A -85,B 0,C 180,E1 -7546.055,E2 -7546.055} C_VEL
LIN {X 0,Y 469.689,Z 440.16,A -85,B 0,C 180,E1 -7547.139,E2 -7547.139} C_VEL
LIN {X 0,Y 469.062,Z 450.385,A -85,B 0,C 180,E1 -7548.33,E2 -7548.33} C_VEL
LIN {X 0,Y 468.571,Z 459.621,A -85,B 0,C 180,E1 -7549.631,E2 -7549.631} C_VEL
LIN {X 0,Y 468.198,Z 467.313,A -85,B 0,C 180,E1 -7550.931,E2 -7550.931} C_VEL
LIN {X 0,Y 467.876,Z 473.704,A -85,B 0,C 180,E1 -7552.23,E2 -7552.23} C_VEL
LIN {X 0,Y 467.665,Z 478.974,A -85,B 0,C 180,E1 -7553.528,E2 -7553.528} C_VEL
LIN {X 0,Y 467.442,Z 484.562,A -85,B 0,C 180,E1 -7555.256,E2 -7555.256} C_VEL
LIN {X 0,Y 467.259,Z 487.695,A -85,B 0,C 180,E1 -7556.551,E2 -7556.551} C_VEL
LIN {X 0,Y 467.192,Z 490.652,A -85,B 0,C 180,E1 -7558.276,E2 -7558.276} C_VEL
LIN {X 0,Y 467.09,Z 492.284,A -85,B 0,C 180,E1 -7560,E2 -7560} C_VEL
LIN {X 0,Y 467.187,Z 492.581,A -85,B 0,C 180,E1 -7561.724,E2 -7561.724} C_VEL
LIN {X 0,Y 467.228,Z 491.581,A -85,B 0,C 180,E1 -7563.449,E2 -7563.449} C_VEL
LIN {X 0,Y 467.367,Z 489.216,A -85,B 0,C 180,E1 -7565.176,E2 -7565.176} C_VEL
LIN {X 0,Y 467.55,Z 486.505,A -85,B 0,C 180,E1 -7566.473,E2 -7566.473} C_VEL
LIN {X 0,Y 467.835,Z 481.605,A -85,B 0,C 180,E1 -7568.205,E2 -7568.205} C_VEL
LIN {X 0,Y 468.015,Z 476.802,A -85,B 0,C 180,E1 -7569.508,E2 -7569.508} C_VEL
LIN {X 0,Y 468.425,Z 469.873,A -85,B 0,C 180,E1 -7571.028,E2 -7571.028} C_VEL
LIN {X 0,Y 468.962,Z 461.285,A -85,B 0,C 180,E1 -7572.54,E2 -7572.54} C_VEL
LIN {X 0,Y 469.54,Z 452.093,A -85,B 0,C 180,E1 -7573.856,E2 -7573.856} C_VEL
LIN {X 0,Y 470.087,Z 441.958,A -85,B 0,C 180,E1 -7575.056,E2 -7575.056} C_VEL
LIN {X 0,Y 470.7,Z 430.748,A -85,B 0,C 180,E1 -7576.146,E2 -7576.146} C_VEL
LIN {X 0,Y 471.274,Z 418.844,A -85,B 0,C 180,E1 -7577.091,E2 -7577.091} C_VEL
LIN {X 0,Y 471.838,Z 406.248,A -85,B 0,C 180,E1 -7577.891,E2 -7577.891} C_VEL
LIN {X 0,Y 471.868,Z 404.271,A -85,B 0,C 180,E1 -7578.002,E2 -7578.002} C_VEL
LIN {X 0,Y 468.391,Z 393.273,A -85,B 0,C 180,E1 -7578.732,E2 -7578.732} C_VEL
LIN {X 0,Y 467.638,Z 390.862,A -85,B 0,C 180,E1 -7578.889,E2 -7578.889} C_VEL
LIN {X 0,Y 467.584,Z 390.87,A -85,B 0,C 180,E1 -7581.268,E2 -7581.268} C_VEL
LIN {X 0,Y 467.577,Z 390.871,A -85,B 0,C 180,E1 -7583.943,E2 -7583.943} C_VEL
LIN {X 0,Y 467.62,Z 390.864,A -85,B 0,C 180,E1 -7586.8,E2 -7586.8} C_VEL
LIN {X 0,Y 467.557,Z 390.871,A -85,B 0,C 180,E1 -7589.738,E2 -7589.738} C_VEL
LIN {X 0,Y 467.586,Z 390.869,A -85,B 0,C 180,E1 -7592.758,E2 -7592.758} C_VEL
LIN {X 0,Y 467.556,Z 390.871,A -85,B 0,C 180,E1 -7595.889,E2 -7595.889} C_VEL
LIN {X 0,Y 467.585,Z 390.868,A -85,B 0,C 180,E1 -7599.144,E2 -7599.144} C_VEL
LIN {X 0,Y 467.589,Z 390.867,A -85,B 0,C 180,E1 -7602.567,E2 -7602.567} C_VEL
LIN {X 0,Y 467.573,Z 390.872,A -85,B 0,C 180,E1 -7605.053,E2 -7605.053} C_VEL
LIN {X 0,Y 467.591,Z 390.945,A -85,B 0,C 180,E1 -7607.615,E2 -7607.615} C_VEL
LIN {X 0,Y 468.859,Z 397.249,A -85,B 0,C 180,E1 -7609.867,E2 -7609.867} C_VEL
LIN {X 0,Y 469.445,Z 401.189,A -85,B 0,C 180,E1 -7611.122,E2 -7611.122} C_VEL
LIN {X 0,Y 469.073,Z 407.38,A -85,B 0,C 180,E1 -7612.862,E2 -7612.862} C_VEL
LIN {X 0,Y 468.373,Z 422.6,A -85,B 0,C 180,E1 -7616.773,E2 -7616.773} C_VEL
LIN {X 0,Y 468.194,Z 435.318,A -85,B 0,C 180,E1 -7619.81,E2 -7619.81} C_VEL
LIN {X 0,Y 467.967,Z 448.42,A -85,B 0,C 180,E1 -7622.801,E2 -7622.801} C_VEL
LIN {X 0,Y 467.826,Z 462.117,A -85,B 0,C 180,E1 -7625.834,E2 -7625.834} C_VEL
LIN {X 0,Y 467.643,Z 477.1,A -85,B 0,C 180,E1 -7629.088,E2 -7629.088} C_VEL
LIN {X 0,Y 467.524,Z 487.673,A -85,B 0,C 180,E1 -7631.361,E2 -7631.361} C_VEL
LIN {X 0,Y 469.185,Z 504.41,A -85,B 0,C 180,E1 -7631.834,E2 -7631.834} C_VEL
LIN {X 0,Y 470.29,Z 514.402,A -85,B 0,C 180,E1 -7632.216,E2 -7632.216} C_VEL
LIN {X 0,Y 470.964,Z 518.847,A -85,B 0,C 180,E1 -7632.411,E2 -7632.411} C_VEL
LIN {X 0,Y 470.364,Z 532.485,A -85,B 0,C 180,E1 -7633.042,E2 -7633.042} C_VEL
LIN {X 0,Y 469.717,Z 545.653,A -85,B 0,C 180,E1 -7633.818,E2 -7633.818} C_VEL
LIN {X 0,Y 469.086,Z 559.014,A -85,B 0,C 180,E1 -7634.799,E2 -7634.799} C_VEL
LIN {X 0,Y 468.499,Z 571.171,A -85,B 0,C 180,E1 -7635.89,E2 -7635.89} C_VEL
LIN {X 0,Y 467.978,Z 582.917,A -85,B 0,C 180,E1 -7637.166,E2 -7637.166} C_VEL
LIN {X 0,Y 467.627,Z 593.133,A -85,B 0,C 180,E1 -7638.513,E2 -7638.513} C_VEL
LIN {X 0,Y 467.293,Z 601.39,A -85,B 0,C 180,E1 -7639.821,E2 -7639.821} C_VEL
LIN {X 0,Y 467.148,Z 609.309,A -85,B 0,C 180,E1 -7641.346,E2 -7641.346} C_VEL
LIN {X 0,Y 466.999,Z 614.843,A -85,B 0,C 180,E1 -7642.65,E2 -7642.65} C_VEL
LIN {X 0,Y 467.017,Z 620.637,A -85,B 0,C 180,E1 -7644.386,E2 -7644.386} C_VEL
LIN {X 0,Y 467.047,Z 623.883,A -85,B 0,C 180,E1 -7645.684,E2 -7645.684} C_VEL
LIN {X 0,Y 466.943,Z 626.87,A -85,B 0,C 180,E1 -7647.411,E2 -7647.411} C_VEL
LIN {X 0,Y 466.881,Z 628.396,A -85,B 0,C 180,E1 -7649.137,E2 -7649.137} C_VEL
LIN {X 0,Y 466.975,Z 628.639,A -85,B 0,C 180,E1 -7649.999,E2 -7649.999} C_VEL
LIN {X 0,Y 466.887,Z 628.01,A -85,B 0,C 180,E1 -7651.724,E2 -7651.724} C_VEL
LIN {X 0,Y 466.918,Z 625.968,A -85,B 0,C 180,E1 -7653.451,E2 -7653.451} C_VEL
LIN {X 0,Y 466.934,Z 622.459,A -85,B 0,C 180,E1 -7655.18,E2 -7655.18} C_VEL
LIN {X 0,Y 466.96,Z 618.381,A -85,B 0,C 180,E1 -7656.618,E2 -7656.618} C_VEL
LIN {X 0,Y 467.033,Z 612.451,A -85,B 0,C 180,E1 -7658.218,E2 -7658.218} C_VEL
LIN {X 0,Y 467.203,Z 605.324,A -85,B 0,C 180,E1 -7659.742,E2 -7659.742} C_VEL
LIN {X 0,Y 467.518,Z 596.502,A -85,B 0,C 180,E1 -7661.268,E2 -7661.268} C_VEL
LIN {X 0,Y 467.934,Z 586.803,A -85,B 0,C 180,E1 -7662.644,E2 -7662.644} C_VEL
LIN {X 0,Y 468.458,Z 576.201,A -85,B 0,C 180,E1 -7663.888,E2 -7663.888} C_VEL
LIN {X 0,Y 469.039,Z 564.974,A -85,B 0,C 180,E1 -7664.978,E2 -7664.978} C_VEL
LIN {X 0,Y 469.733,Z 552.677,A -85,B 0,C 180,E1 -7665.956,E2 -7665.956} C_VEL
LIN {X 0,Y 470.411,Z 539.906,A -85,B 0,C 180,E1 -7666.776,E2 -7666.776} C_VEL
LIN {X 0,Y 471.034,Z 526.004,A -85,B 0,C 180,E1 -7667.473,E2 -7667.473} C_VEL
LIN {X 0,Y 471.117,Z 517.82,A -85,B 0,C 180,E1 -7667.806,E2 -7667.806} C_VEL
LIN {X 0,Y 469.347,Z 505.095,A -85,B 0,C 180,E1 -7668.27,E2 -7668.27} C_VEL
LIN {X 0,Y 467.626,Z 492.751,A -85,B 0,C 180,E1 -7668.615,E2 -7668.615} C_VEL
LIN {X 0,Y 468.003,Z 477.991,A -85,B 0,C 180,E1 -7672.049,E2 -7672.049} C_VEL
LIN {X 0,Y 468.457,Z 464.243,A -85,B 0,C 180,E1 -7675.312,E2 -7675.312} C_VEL
LIN {X 0,Y 468.857,Z 452.35,A -85,B 0,C 180,E1 -7678.189,E2 -7678.189} C_VEL
LIN {X 0,Y 469.41,Z 440.891,A -85,B 0,C 180,E1 -7681.017,E2 -7681.017} C_VEL
LIN {X 0,Y 469.999,Z 428.704,A -85,B 0,C 180,E1 -7684.106,E2 -7684.106} C_VEL
LIN {X 0,Y 470.829,Z 414.815,A -85,B 0,C 180,E1 -7687.733,E2 -7687.733} C_VEL
LIN {X 0,Y 471.053,Z 408.391,A -85,B 0,C 180,E1 -7689.466,E2 -7689.466} C_VEL
LIN {X 0,Y 469.795,Z 401.158,A -85,B 0,C 180,E1 -7691.584,E2 -7691.584} C_VEL
LIN {X 0,Y 467.585,Z 390.867,A -85,B 0,C 180,E1 -7694.796,E2 -7694.796} C_VEL
LIN {X 0,Y 467.616,Z 390.863,A -85,B 0,C 180,E1 -7697.443,E2 -7697.443} C_VEL
LIN {X 0,Y 467.616,Z 390.86,A -85,B 0,C 180,E1 -7700.859,E2 -7700.859} C_VEL
LIN {X 0,Y 467.554,Z 390.868,A -85,B 0,C 180,E1 -7704.259,E2 -7704.259} C_VEL
LIN {X 0,Y 467.573,Z 390.869,A -85,B 0,C 180,E1 -7707.32,E2 -7707.32} C_VEL
LIN {X 0,Y 467.568,Z 390.866,A -85,B 0,C 180,E1 -7710.665,E2 -7710.665} C_VEL
LIN {X 0,Y 467.618,Z 390.862,A -85,B 0,C 180,E1 -7713.2,E2 -7713.2} C_VEL
LIN {X 0,Y 467.582,Z 390.864,A -85,B 0,C 180,E1 -7716.468,E2 -7716.468} C_VEL
LIN {X 0,Y 467.613,Z 390.862,A -85,B 0,C 180,E1 -7719.777,E2 -7719.777} C_VEL
LIN {X 0,Y 467.599,Z 390.862,A -85,B 0,C 180,E1 -7722.507,E2 -7722.507} C_VEL
LIN {X 0,Y 467.599,Z 390.866,A -85,B 0,C 180,E1 -7725.196,E2 -7725.196} C_VEL
LIN {X 0,Y 467.672,Z 390.854,A -85,B 0,C 180,E1 -7727.855,E2 -7727.855} C_VEL
LIN {X 0,Y 467.672,Z 390.857,A -85,B 0,C 180,E1 -7731.357,E2 -7731.357} C_VEL
LIN {X 0,Y 467.734,Z 390.846,A -85,B 0,C 180,E1 -7733.963,E2 -7733.963} C_VEL
LIN {X 0,Y 467.851,Z 390.834,A -85,B 0,C 180,E1 -7737.417,E2 -7737.417} C_VEL
LIN {X 0,Y 467.872,Z 390.829,A -85,B 0,C 180,E1 -7740,E2 -7740} C_VEL
LIN {X 0,Y 467.851,Z 390.831,A -85,B 0,C 180,E1 -7742.583,E2 -7742.583} C_VEL
LIN {X 0,Y 467.737,Z 390.846,A -85,B 0,C 180,E1 -7746.038,E2 -7746.038} C_VEL
LIN {X 0,Y 467.672,Z 390.854,A -85,B 0,C 180,E1 -7748.643,E2 -7748.643} C_VEL
LIN {X 0,Y 467.681,Z 390.852,A -85,B 0,C 180,E1 -7752.379,E2 -7752.379} C_VEL
LIN {X 0,Y 467.639,Z 390.858,A -85,B 0,C 180,E1 -7755.886,E2 -7755.886} C_VEL
LIN {X 0,Y 467.615,Z 390.863,A -85,B 0,C 180,E1 -7759.308,E2 -7759.308} C_VEL
LIN {X 0,Y 467.527,Z 390.872,A -85,B 0,C 180,E1 -7762.075,E2 -7762.075} C_VEL
LIN {X 0,Y 467.595,Z 390.866,A -85,B 0,C 180,E1 -7764.888,E2 -7764.888} C_VEL
LIN {X 0,Y 467.619,Z 390.861,A -85,B 0,C 180,E1 -7767.769,E2 -7767.769} C_VEL
LIN {X 0,Y 467.561,Z 390.871,A -85,B 0,C 180,E1 -7771.046,E2 -7771.046} C_VEL
LIN {X 0,Y 467.583,Z 390.864,A -85,B 0,C 180,E1 -7774.244,E2 -7774.244} C_VEL
LIN {X 0,Y 467.544,Z 390.871,A -85,B 0,C 180,E1 -7777.188,E2 -7777.188} C_VEL
LIN {X 0,Y 467.573,Z 390.866,A -85,B 0,C 180,E1 -7780.266,E2 -7780.266} C_VEL
LIN {X 0,Y 467.581,Z 390.866,A -85,B 0,C 180,E1 -7782.568,E2 -7782.568} C_VEL
LIN {X 0,Y 467.566,Z 390.869,A -85,B 0,C 180,E1 -7785.054,E2 -7785.054} C_VEL
LIN {X 0,Y 467.584,Z 390.865,A -85,B 0,C 180,E1 -7787.441,E2 -7787.441} C_VEL
LIN {X 0,Y 467.615,Z 390.864,A -85,B 0,C 180,E1 -7790.86,E2 -7790.86} C_VEL
LIN {X 0,Y 467.561,Z 390.867,A -85,B 0,C 180,E1 -7794.262,E2 -7794.262} C_VEL
LIN {X 0,Y 467.581,Z 390.866,A -85,B 0,C 180,E1 -7797.322,E2 -7797.322} C_VEL
LIN {X 0,Y 467.57,Z 390.87,A -85,B 0,C 180,E1 -7800.669,E2 -7800.669} C_VEL
LIN {X 0,Y 467.616,Z 390.861,A -85,B 0,C 180,E1 -7803.201,E2 -7803.201} C_VEL
LIN {X 0,Y 467.593,Z 390.865,A -85,B 0,C 180,E1 -7806.47,E2 -7806.47} C_VEL
LIN {X 0,Y 467.624,Z 390.86,A -85,B 0,C 180,E1 -7809.778,E2 -7809.778} C_VEL
LIN {X 0,Y 467.605,Z 390.864,A -85,B 0,C 180,E1 -7812.508,E2 -7812.508} C_VEL
LIN {X 0,Y 467.533,Z 390.874,A -85,B 0,C 180,E1 -7815.195,E2 -7815.195} C_VEL
LIN {X 0,Y 467.509,Z 390.876,A -85,B 0,C 180,E1 -7815.432,E2 -7815.432} C_VEL
LIN {X 0,Y 466.787,Z 390.967,A -85,B 0,C 180,E1 -7815.78,E2 -7815.78} C_VEL
LIN {X 0,Y 461.058,Z 391.682,A -85,B 0,C 180,E1 -7816.807,E2 -7816.807} C_VEL
LIN {X 0,Y 460.348,Z 391.771,A -85,B 0,C 180,E1 -7817.163,E2 -7817.163} C_VEL
LIN {X 0,Y 460.333,Z 391.775,A -85,B 0,C 180,E1 -7817.522,E2 -7817.522} C_VEL
LIN {X 0,Y 463.872,Z 403.355,A -85,B 0,C 180,E1 -7817.978,E2 -7817.978} C_VEL
LIN {X 0,Y 463.712,Z 414.752,A -85,B 0,C 180,E1 -7818.448,E2 -7818.448} C_VEL
LIN {X 0,Y 463.416,Z 426.023,A -85,B 0,C 180,E1 -7819.073,E2 -7819.073} C_VEL
LIN {X 0,Y 463.042,Z 436.742,A -85,B 0,C 180,E1 -7819.838,E2 -7819.838} C_VEL
LIN {X 0,Y 462.514,Z 447.722,A -85,B 0,C 180,E1 -7820.821,E2 -7820.821} C_VEL
LIN {X 0,Y 462.036,Z 457.322,A -85,B 0,C 180,E1 -7821.893,E2 -7821.893} C_VEL
LIN {X 0,Y 461.628,Z 465.407,A -85,B 0,C 180,E1 -7823.005,E2 -7823.005} C_VEL
LIN {X 0,Y 461.284,Z 473.162,A -85,B 0,C 180,E1 -7824.318,E2 -7824.318} C_VEL
LIN {X 0,Y 460.921,Z 479.422,A -85,B 0,C 180,E1 -7825.629,E2 -7825.629} C_VEL
LIN {X 0,Y 460.63,Z 484.396,A -85,B 0,C 180,E1 -7826.94,E2 -7826.94} C_VEL
LIN {X 0,Y 460.452,Z 488.235,A -85,B 0,C 180,E1 -7828.252,E2 -7828.252} C_VEL
LIN {X 0,Y 460.335,Z 490.216,A -85,B 0,C 180,E1 -7829.126,E2 -7829.126} C_VEL
LIN {X 0,Y 460.133,Z 492.981,A -85,B 0,C 180,E1 -7830.876,E2 -7830.876} C_VEL
LIN {X 0,Y 460.196,Z 493.749,A -85,B 0,C 180,E1 -7831.751,E2 -7831.751} C_VEL
LIN {X 0,Y 460.146,Z 494.134,A -85,B 0,C 180,E1 -7833.503,E2 -7833.503} C_VEL
LIN {X 0,Y 460.197,Z 493.765,A -85,B 0,C 180,E1 -7834.38,E2 -7834.38} C_VEL
LIN {X 0,Y 460.316,Z 492.976,A -85,B 0,C 180,E1 -7835.257,E2 -7835.257} C_VEL
LIN {X 0,Y 460.399,Z 490.233,A -85,B 0,C 180,E1 -7837.015,E2 -7837.015} C_VEL
LIN {X 0,Y 460.553,Z 487.056,A -85,B 0,C 180,E1 -7838.336,E2 -7838.336} C_VEL
LIN {X 0,Y 460.842,Z 482.815,A -85,B 0,C 180,E1 -7839.658,E2 -7839.658} C_VEL
LIN {X 0,Y 461.177,Z 476.349,A -85,B 0,C 180,E1 -7841.205,E2 -7841.205} C_VEL
LIN {X 0,Y 461.498,Z 469.234,A -85,B 0,C 180,E1 -7842.541,E2 -7842.541} C_VEL
LIN {X 0,Y 462.027,Z 460.41,A -85,B 0,C 180,E1 -7843.862,E2 -7843.862} C_VEL
LIN {X 0,Y 462.523,Z 450.158,A -85,B 0,C 180,E1 -7845.083,E2 -7845.083} C_VEL
LIN {X 0,Y 463.027,Z 439.688,A -85,B 0,C 180,E1 -7846.082,E2 -7846.082} C_VEL
LIN {X 0,Y 463.461,Z 429.159,A -85,B 0,C 180,E1 -7846.879,E2 -7846.879} C_VEL
LIN {X 0,Y 463.808,Z 417.684,A -85,B 0,C 180,E1 -7847.562,E2 -7847.562} C_VEL
LIN {X 0,Y 464.099,Z 405.179,A -85,B 0,C 180,E1 -7848.115,E2 -7848.115} C_VEL
LIN {X 0,Y 463.537,Z 402.038,A -85,B 0,C 180,E1 -7848.246,E2 -7848.246} C_VEL
LIN {X 0,Y 460.309,Z 391.775,A -85,B 0,C 180,E1 -7848.66,E2 -7848.66} C_VEL
LIN {X 0,Y 460.477,Z 391.752,A -85,B 0,C 180,E1 -7851.488,E2 -7851.488} C_VEL
LIN {X 0,Y 460.548,Z 391.74,A -85,B 0,C 180,E1 -7854.333,E2 -7854.333} C_VEL
LIN {X 0,Y 460.58,Z 391.74,A -85,B 0,C 180,E1 -7857.244,E2 -7857.244} C_VEL
LIN {X 0,Y 460.517,Z 391.746,A -85,B 0,C 180,E1 -7860.24,E2 -7860.24} C_VEL
LIN {X 0,Y 460.525,Z 391.746,A -85,B 0,C 180,E1 -7863.326,E2 -7863.326} C_VEL
LIN {X 0,Y 460.482,Z 391.754,A -85,B 0,C 180,E1 -7866.53,E2 -7866.53} C_VEL
LIN {X 0,Y 460.532,Z 391.739,A -85,B 0,C 180,E1 -7869.863,E2 -7869.863} C_VEL
LIN {X 0,Y 460.519,Z 391.745,A -85,B 0,C 180,E1 -7872.9,E2 -7872.9} C_VEL
LIN {X 0,Y 460.525,Z 391.741,A -85,B 0,C 180,E1 -7875.829,E2 -7875.829} C_VEL
LIN {X 0,Y 460.539,Z 391.737,A -85,B 0,C 180,E1 -7878.989,E2 -7878.989} C_VEL
LIN {X 0,Y 460.531,Z 391.724,A -85,B 0,C 180,E1 -7881.267,E2 -7881.267} C_VEL
LIN {X 0,Y 460.518,Z 391.745,A -85,B 0,C 180,E1 -7884.555,E2 -7884.555} C_VEL
LIN {X 0,Y 460.536,Z 391.741,A -85,B 0,C 180,E1 -7887.716,E2 -7887.716} C_VEL
LIN {X 0,Y 460.543,Z 391.719,A -85,B 0,C 180,E1 -7890.769,E2 -7890.769} C_VEL
LIN {X 0,Y 460.56,Z 391.738,A -85,B 0,C 180,E1 -7893.734,E2 -7893.734} C_VEL
LIN {X 0,Y 460.549,Z 391.739,A -85,B 0,C 180,E1 -7896.624,E2 -7896.624} C_VEL
LIN {X 0,Y 460.555,Z 391.744,A -85,B 0,C 180,E1 -7899.453,E2 -7899.453} C_VEL
LIN {X 0,Y 460.553,Z 391.741,A -85,B 0,C 180,E1 -7902.23,E2 -7902.23} C_VEL
LIN {X 0,Y 460.553,Z 391.744,A -85,B 0,C 180,E1 -7903.193,E2 -7903.193} C_VEL
LIN {X 0,Y 464.546,Z 404.912,A -85,B 0,C 180,E1 -7904.057,E2 -7904.057} C_VEL
LIN {X 0,Y 464.039,Z 417.283,A -85,B 0,C 180,E1 -7904.855,E2 -7904.855} C_VEL
LIN {X 0,Y 463.448,Z 429.682,A -85,B 0,C 180,E1 -7905.846,E2 -7905.846} C_VEL
LIN {X 0,Y 462.834,Z 440.956,A -85,B 0,C 180,E1 -7906.946,E2 -7906.946} C_VEL
LIN {X 0,Y 462.168,Z 451.216,A -85,B 0,C 180,E1 -7908.153,E2 -7908.153} C_VEL
LIN {X 0,Y 461.649,Z 460.484,A -85,B 0,C 180,E1 -7909.474,E2 -7909.474} C_VEL
LIN {X 0,Y 461.258,Z 468.203,A -85,B 0,C 180,E1 -7910.794,E2 -7910.794} C_VEL
LIN {X 0,Y 460.914,Z 474.621,A -85,B 0,C 180,E1 -7912.112,E2 -7912.112} C_VEL
LIN {X 0,Y 460.684,Z 479.918,A -85,B 0,C 180,E1 -7913.43,E2 -7913.43} C_VEL
LIN {X 0,Y 460.441,Z 485.535,A -85,B 0,C 180,E1 -7915.184,E2 -7915.184} C_VEL
LIN {X 0,Y 460.243,Z 488.688,A -85,B 0,C 180,E1 -7916.498,E2 -7916.498} C_VEL
LIN {X 0,Y 460.179,Z 491.671,A -85,B 0,C 180,E1 -7918.249,E2 -7918.249} C_VEL
LIN {X 0,Y 460.071,Z 493.321,A -85,B 0,C 180,E1 -7920,E2 -7920} C_VEL
LIN {X 0,Y 460.175,Z 493.631,A -85,B 0,C 180,E1 -7921.75,E2 -7921.75} C_VEL
LIN {X 0,Y 460.217,Z 492.637,A -85,B 0,C 180,E1 -7923.502,E2 -7923.502} C_VEL
LIN {X 0,Y 460.374,Z 490.268,A -85,B 0,C 180,E1 -7925.255,E2 -7925.255} C_VEL
LIN {X 0,Y 460.583,Z 487.562,A -85,B 0,C 180,E1 -7926.571,E2 -7926.571} C_VEL
LIN {X 0,Y 460.88,Z 482.676,A -85,B 0,C 180,E1 -7928.329,E2 -7928.329} C_VEL
LIN {X 0,Y 461.092,Z 477.893,A -85,B 0,C 180,E1 -7929.652,E2 -7929.652} C_VEL
LIN {X 0,Y 461.551,Z 470.982,A -85,B 0,C 180,E1 -7931.195,E2 -7931.195} C_VEL
LIN {X 0,Y 462.128,Z 462.374,A -85,B 0,C 180,E1 -7932.729,E2 -7932.729} C_VEL
LIN {X 0,Y 462.729,Z 453.169,A -85,B 0,C 180,E1 -7934.064,E2 -7934.064} C_VEL
LIN {X 0,Y 463.316,Z 443.019,A -85,B 0,C 180,E1 -7935.281,E2 -7935.281} C_VEL
LIN {X 0,Y 463.966,Z 431.845,A -85,B 0,C 180,E1 -7936.387,E2 -7936.387} C_VEL
LIN {X 0,Y 464.582,Z 420.013,A -85,B 0,C 180,E1 -7937.345,E2 -7937.345} C_VEL
LIN {X 0,Y 465.201,Z 407.523,A -85,B 0,C 180,E1 -7938.155,E2 -7938.155} C_VEL
LIN {X 0,Y 464.769,Z 404.346,A -85,B 0,C 180,E1 -7938.358,E2 -7938.358} C_VEL
LIN {X 0,Y 460.593,Z 391.74,A -85,B 0,C 180,E1 -7939.209,E2 -7939.209} C_VEL
LIN {X 0,Y 460.515,Z 391.751,A -85,B 0,C 180,E1 -7942.428,E2 -7942.428} C_VEL
LIN {X 0,Y 460.571,Z 391.742,A -85,B 0,C 180,E1 -7945.802,E2 -7945.802} C_VEL
LIN {X 0,Y 460.555,Z 391.742,A -85,B 0,C 180,E1 -7948.233,E2 -7948.233} C_VEL
LIN {X 0,Y 460.524,Z 391.748,A -85,B 0,C 180,E1 -7951.283,E2 -7951.283} C_VEL
LIN {X 0,Y 460.534,Z 391.746,A -85,B 0,C 180,E1 -7954.505,E2 -7954.505} C_VEL
LIN {X 0,Y 460.504,Z 391.75,A -85,B 0,C 180,E1 -7957.623,E2 -7957.623} C_VEL
LIN {X 0,Y 460.545,Z 391.745,A -85,B 0,C 180,E1 -7960.269,E2 -7960.269} C_VEL
LIN {X 0,Y 460.503,Z 391.75,A -85,B 0,C 180,E1 -7963.375,E2 -7963.375} C_VEL
LIN {X 0,Y 460.503,Z 391.754,A -85,B 0,C 180,E1 -7966.624,E2 -7966.624} C_VEL
LIN {X 0,Y 460.544,Z 391.861,A -85,B 0,C 180,E1 -7967.196,E2 -7967.196} C_VEL
LIN {X 0,Y 461.825,Z 398.131,A -85,B 0,C 180,E1 -7969.543,E2 -7969.543} C_VEL
LIN {X 0,Y 462.532,Z 403.009,A -85,B 0,C 180,E1 -7971.139,E2 -7971.139} C_VEL
LIN {X 0,Y 462.213,Z 407.843,A -85,B 0,C 180,E1 -7972.54,E2 -7972.54} C_VEL
LIN {X 0,Y 461.407,Z 421.719,A -85,B 0,C 180,E1 -7976.223,E2 -7976.223} C_VEL
LIN {X 0,Y 461.159,Z 434.205,A -85,B 0,C 180,E1 -7979.3,E2 -7979.3} C_VEL
LIN {X 0,Y 460.988,Z 444.801,A -85,B 0,C 180,E1 -7981.795,E2 -7981.795} C_VEL
LIN {X 0,Y 460.808,Z 458.703,A -85,B 0,C 180,E1 -7984.961,E2 -7984.961} C_VEL
LIN {X 0,Y 460.616,Z 473.643,A -85,B 0,C 180,E1 -7988.283,E2 -7988.283} C_VEL
LIN {X 0,Y 460.449,Z 486.353,A -85,B 0,C 180,E1 -7991.042,E2 -7991.042} C_VEL
LIN {X 0,Y 462.195,Z 502.086,A -85,B 0,C 180,E1 -7991.507,E2 -7991.507} C_VEL
LIN {X 0,Y 463.218,Z 514.413,A -85,B 0,C 180,E1 -7991.982,E2 -7991.982} C_VEL
LIN {X 0,Y 464.015,Z 520.151,A -85,B 0,C 180,E1 -7992.252,E2 -7992.252} C_VEL
LIN {X 0,Y 463.332,Z 534.778,A -85,B 0,C 180,E1 -7992.984,E2 -7992.984} C_VEL
LIN {X 0,Y 462.662,Z 547.524,A -85,B 0,C 180,E1 -7993.791,E2 -7993.791} C_VEL
LIN {X 0,Y 462.014,Z 560.315,A -85,B 0,C 180,E1 -7994.787,E2 -7994.787} C_VEL
LIN {X 0,Y 461.377,Z 572.015,A -85,B 0,C 180,E1 -7995.893,E2 -7995.893} C_VEL
LIN {X 0,Y 460.887,Z 583.565,A -85,B 0,C 180,E1 -7997.216,E2 -7997.216} C_VEL
LIN {X 0,Y 460.51,Z 593.287,A -85,B 0,C 180,E1 -7998.556,E2 -7998.556} C_VEL
LIN {X 0,Y 460.201,Z 601.347,A -85,B 0,C 180,E1 -7999.884,E2 -7999.884} C_VEL
LIN {X 0,Y 460.081,Z 608.107,A -85,B 0,C 180,E1 -8001.212,E2 -8001.212} C_VEL
LIN {X 0,Y 459.936,Z 613.677,A -85,B 0,C 180,E1 -8002.536,E2 -8002.536} C_VEL
LIN {X 0,Y 459.937,Z 618.197,A -85,B 0,C 180,E1 -8003.859,E2 -8003.859} C_VEL
LIN {X 0,Y 459.99,Z 621.807,A -85,B 0,C 180,E1 -8005.179,E2 -8005.179} C_VEL
LIN {X 0,Y 459.933,Z 624.495,A -85,B 0,C 180,E1 -8006.495,E2 -8006.495} C_VEL
LIN {X 0,Y 459.883,Z 626.78,A -85,B 0,C 180,E1 -8008.248,E2 -8008.248} C_VEL
LIN {X 0,Y 459.962,Z 627.629,A -85,B 0,C 180,E1 -8009.999,E2 -8009.999} C_VEL
LIN {X 0,Y 459.852,Z 627.011,A -85,B 0,C 180,E1 -8011.751,E2 -8011.751} C_VEL
LIN {X 0,Y 459.876,Z 624.98,A -85,B 0,C 180,E1 -8013.504,E2 -8013.504} C_VEL
LIN {X 0,Y 459.868,Z 621.47,A -85,B 0,C 180,E1 -8015.26,E2 -8015.26} C_VEL
LIN {X 0,Y 459.899,Z 617.677,A -85,B 0,C 180,E1 -8016.634,E2 -8016.634} C_VEL
LIN {X 0,Y 459.956,Z 611.451,A -85,B 0,C 180,E1 -8018.345,E2 -8018.345} C_VEL
LIN {X 0,Y 460.127,Z 604.313,A -85,B 0,C 180,E1 -8019.893,E2 -8019.893} C_VEL
LIN {X 0,Y 460.489,Z 595.484,A -85,B 0,C 180,E1 -8021.443,E2 -8021.443} C_VEL
LIN {X 0,Y 460.894,Z 586.235,A -85,B 0,C 180,E1 -8022.776,E2 -8022.776} C_VEL
LIN {X 0,Y 461.473,Z 575.14,A -85,B 0,C 180,E1 -8024.102,E2 -8024.102} C_VEL
LIN {X 0,Y 462.075,Z 563.876,A -85,B 0,C 180,E1 -8025.209,E2 -8025.209} C_VEL
LIN {X 0,Y 462.847,Z 551.547,A -85,B 0,C 180,E1 -8026.2,E2 -8026.2} C_VEL
LIN {X 0,Y 463.565,Z 538.134,A -85,B 0,C 180,E1 -8027.066,E2 -8027.066} C_VEL
LIN {X 0,Y 464.175,Z 524.782,A -85,B 0,C 180,E1 -8027.739,E2 -8027.739} C_VEL
LIN {X 0,Y 464.213,Z 518.751,A -85,B 0,C 180,E1 -8027.994,E2 -8027.994} C_VEL
LIN {X 0,Y 462.383,Z 504.8,A -85,B 0,C 180,E1 -8028.527,E2 -8028.527} C_VEL
LIN {X 0,Y 460.583,Z 491.924,A -85,B 0,C 180,E1 -8028.906,E2 -8028.906} C_VEL
LIN {X 0,Y 460.976,Z 477.184,A -85,B 0,C 180,E1 -8032.404,E2 -8032.404} C_VEL
LIN {X 0,Y 461.444,Z 463.761,A -85,B 0,C 180,E1 -8035.647,E2 -8035.647} C_VEL
LIN {X 0,Y 461.894,Z 451.628,A -85,B 0,C 180,E1 -8038.638,E2 -8038.638} C_VEL
LIN {X 0,Y 462.427,Z 441.79,A -85,B 0,C 180,E1 -8041.112,E2 -8041.112} C_VEL
LIN {X 0,Y 463.027,Z 429.919,A -85,B 0,C 180,E1 -8044.165,E2 -8044.165} C_VEL
LIN {X 0,Y 463.946,Z 415.365,A -85,B 0,C 180,E1 -8048.028,E2 -8048.028} C_VEL
LIN {X 0,Y 464.161,Z 410.049,A -85,B 0,C 180,E1 -8049.488,E2 -8049.488} C_VEL
LIN {X 0,Y 462.697,Z 401.805,A -85,B 0,C 180,E1 -8051.936,E2 -8051.936} C_VEL
LIN {X 0,Y 460.514,Z 391.748,A -85,B 0,C 180,E1 -8055.126,E2 -8055.126} C_VEL
LIN {X 0,Y 460.538,Z 391.743,A -85,B 0,C 180,E1 -8058.395,E2 -8058.395} C_VEL
LIN {X 0,Y 460.541,Z 391.744,A -85,B 0,C 180,E1 -8061.269,E2 -8061.269} C_VEL
LIN {X 0,Y 460.505,Z 391.746,A -85,B 0,C 180,E1 -8064.554,E2 -8064.554} C_VEL
LIN {X 0,Y 460.523,Z 391.746,A -85,B 0,C 180,E1 -8067.715,E2 -8067.715} C_VEL
LIN {X 0,Y 460.538,Z 391.742,A -85,B 0,C 180,E1 -8070.769,E2 -8070.769} C_VEL
LIN {X 0,Y 460.558,Z 391.741,A -85,B 0,C 180,E1 -8073.735,E2 -8073.735} C_VEL
LIN {X 0,Y 460.535,Z 391.742,A -85,B 0,C 180,E1 -8076.624,E2 -8076.624} C_VEL
LIN {X 0,Y 460.542,Z 391.745,A -85,B 0,C 180,E1 -8079.452,E2 -8079.452} C_VEL
LIN {X 0,Y 460.549,Z 391.741,A -85,B 0,C 180,E1 -8082.23,E2 -8082.23} C_VEL
LIN {X 0,Y 460.557,Z 391.741,A -85,B 0,C 180,E1 -8084.965,E2 -8084.965} C_VEL
LIN {X 0,Y 460.618,Z 391.733,A -85,B 0,C 180,E1 -8087.666,E2 -8087.666} C_VEL
LIN {X 0,Y 460.619,Z 391.736,A -85,B 0,C 180,E1 -8091.224,E2 -8091.224} C_VEL
LIN {X 0,Y 460.7,Z 391.722,A -85,B 0,C 180,E1 -8093.87,E2 -8093.87} C_VEL
LIN {X 0,Y 460.816,Z 391.71,A -85,B 0,C 180,E1 -8097.378,E2 -8097.378} C_VEL
LIN {X 0,Y 460.843,Z 391.704,A -85,B 0,C 180,E1 -8100,E2 -8100} C_VEL
LIN {X 0,Y 460.816,Z 391.708,A -85,B 0,C 180,E1 -8102.623,E2 -8102.623} C_VEL
LIN {X 0,Y 460.703,Z 391.722,A -85,B 0,C 180,E1 -8106.13,E2 -8106.13} C_VEL
LIN {X 0,Y 460.62,Z 391.733,A -85,B 0,C 180,E1 -8108.777,E2 -8108.777} C_VEL
LIN {X 0,Y 460.624,Z 391.731,A -85,B 0,C 180,E1 -8112.457,E2 -8112.457} C_VEL
LIN {X 0,Y 460.59,Z 391.736,A -85,B 0,C 180,E1 -8115.998,E2 -8115.998} C_VEL
LIN {X 0,Y 460.561,Z 391.742,A -85,B 0,C 180,E1 -8118.903,E2 -8118.903} C_VEL
LIN {X 0,Y 460.506,Z 391.747,A -85,B 0,C 180,E1 -8121.486,E2 -8121.486} C_VEL
LIN {X 0,Y 460.534,Z 391.743,A -85,B 0,C 180,E1 -8124.333,E2 -8124.333} C_VEL
LIN {X 0,Y 460.575,Z 391.739,A -85,B 0,C 180,E1 -8127.244,E2 -8127.244} C_VEL
LIN {X 0,Y 460.503,Z 391.746,A -85,B 0,C 180,E1 -8130.241,E2 -8130.241} C_VEL
LIN {X 0,Y 460.522,Z 391.745,A -85,B 0,C 180,E1 -8133.326,E2 -8133.326} C_VEL
LIN {X 0,Y 460.472,Z 391.751,A -85,B 0,C 180,E1 -8136.53,E2 -8136.53} C_VEL
LIN {X 0,Y 460.552,Z 391.741,A -85,B 0,C 180,E1 -8139.861,E2 -8139.861} C_VEL
LIN {X 0,Y 460.513,Z 391.749,A -85,B 0,C 180,E1 -8142.902,E2 -8142.902} C_VEL
LIN {X 0,Y 460.507,Z 391.747,A -85,B 0,C 180,E1 -8145.832,E2 -8145.832} C_VEL
LIN {X 0,Y 460.535,Z 391.745,A -85,B 0,C 180,E1 -8148.991,E2 -8148.991} C_VEL
LIN {X 0,Y 460.544,Z 391.742,A -85,B 0,C 180,E1 -8151.27,E2 -8151.27} C_VEL
LIN {X 0,Y 460.511,Z 391.747,A -85,B 0,C 180,E1 -8154.556,E2 -8154.556} C_VEL
LIN {X 0,Y 460.53,Z 391.744,A -85,B 0,C 180,E1 -8157.717,E2 -8157.717} C_VEL
LIN {X 0,Y 460.539,Z 391.746,A -85,B 0,C 180,E1 -8160.77,E2 -8160.77} C_VEL
LIN {X 0,Y 460.563,Z 391.74,A -85,B 0,C 180,E1 -8163.736,E2 -8163.736} C_VEL
LIN {X 0,Y 460.546,Z 391.745,A -85,B 0,C 180,E1 -8166.625,E2 -8166.625} C_VEL
LIN {X 0,Y 460.552,Z 391.741,A -85,B 0,C 180,E1 -8169.454,E2 -8169.454} C_VEL
LIN {X 0,Y 460.557,Z 391.741,A -85,B 0,C 180,E1 -8172.231,E2 -8172.231} C_VEL
LIN {X 0,Y 460.508,Z 391.748,A -85,B 0,C 180,E1 -8174.964,E2 -8174.964} C_VEL
LIN {X 0,Y 460.348,Z 391.771,A -85,B 0,C 180,E1 -8177.163,E2 -8177.163} C_VEL
LIN {X 0,Y 460.336,Z 392.611,A -85,B 0,C 180,E1 -8177.389,E2 -8177.389} C_VEL
LIN {X 0,Y 460.32,Z 394.94,A -85,B 0,C 180,E1 -8177.573,E2 -8177.573} C_VEL
LIN {X 0,Y 459.87,Z 406.452,A -85,B 0,C 180,E1 -8177.945,E2 -8177.945} C_VEL
LIN {X 0,Y 457.229,Z 418.058,A -85,B 0,C 180,E1 -8178.35,E2 -8178.35} C_VEL
LIN {X 0,Y 456.712,Z 421.473,A -85,B 0,C 180,E1 -8178.539,E2 -8178.539} C_VEL
LIN {X 0,Y 456.31,Z 433.887,A -85,B 0,C 180,E1 -8179.35,E2 -8179.35} C_VEL
LIN {X 0,Y 455.859,Z 444.52,A -85,B 0,C 180,E1 -8180.237,E2 -8180.237} C_VEL
LIN {X 0,Y 455.318,Z 454.721,A -85,B 0,C 180,E1 -8181.301,E2 -8181.301} C_VEL
LIN {X 0,Y 454.88,Z 463.634,A -85,B 0,C 180,E1 -8182.455,E2 -8182.455} C_VEL
LIN {X 0,Y 454.361,Z 471.993,A -85,B 0,C 180,E1 -8183.785,E2 -8183.785} C_VEL
LIN {X 0,Y 453.995,Z 478.655,A -85,B 0,C 180,E1 -8185.117,E2 -8185.117} C_VEL
LIN {X 0,Y 453.728,Z 483.976,A -85,B 0,C 180,E1 -8186.449,E2 -8186.449} C_VEL
LIN {X 0,Y 453.552,Z 488.138,A -85,B 0,C 180,E1 -8187.781,E2 -8187.781} C_VEL
LIN {X 0,Y 453.325,Z 491.285,A -85,B 0,C 180,E1 -8189.113,E2 -8189.113} C_VEL
LIN {X 0,Y 453.112,Z 494.027,A -85,B 0,C 180,E1 -8190.89,E2 -8190.89} C_VEL
LIN {X 0,Y 453.178,Z 494.77,A -85,B 0,C 180,E1 -8191.778,E2 -8191.778} C_VEL
LIN {X 0,Y 453.121,Z 495.132,A -85,B 0,C 180,E1 -8193.558,E2 -8193.558} C_VEL
LIN {X 0,Y 453.179,Z 494.75,A -85,B 0,C 180,E1 -8194.448,E2 -8194.448} C_VEL
LIN {X 0,Y 453.312,Z 493.937,A -85,B 0,C 180,E1 -8195.338,E2 -8195.338} C_VEL
LIN {X 0,Y 453.405,Z 491.17,A -85,B 0,C 180,E1 -8197.124,E2 -8197.124} C_VEL
LIN {X 0,Y 453.573,Z 487.967,A -85,B 0,C 180,E1 -8198.466,E2 -8198.466} C_VEL
LIN {X 0,Y 453.897,Z 483.695,A -85,B 0,C 180,E1 -8199.807,E2 -8199.807} C_VEL
LIN {X 0,Y 454.251,Z 477.182,A -85,B 0,C 180,E1 -8201.378,E2 -8201.378} C_VEL
LIN {X 0,Y 454.599,Z 470.113,A -85,B 0,C 180,E1 -8202.72,E2 -8202.72} C_VEL
LIN {X 0,Y 455.092,Z 462.77,A -85,B 0,C 180,E1 -8203.85,E2 -8203.85} C_VEL
LIN {X 0,Y 455.558,Z 453.913,A -85,B 0,C 180,E1 -8204.976,E2 -8204.976} C_VEL
LIN {X 0,Y 456.044,Z 444.044,A -85,B 0,C 180,E1 -8205.991,E2 -8205.991} C_VEL
LIN {X 0,Y 456.541,Z 433.115,A -85,B 0,C 180,E1 -8206.892,E2 -8206.892} C_VEL
LIN {X 0,Y 456.957,Z 421.72,A -85,B 0,C 180,E1 -8207.631,E2 -8207.631} C_VEL
LIN {X 0,Y 457.225,Z 409.036,A -85,B 0,C 180,E1 -8208.244,E2 -8208.244} C_VEL
LIN {X 0,Y 457.194,Z 404.994,A -85,B 0,C 180,E1 -8208.404,E2 -8208.404} C_VEL
LIN {X 0,Y 453.259,Z 392.653,A -85,B 0,C 180,E1 -8208.943,E2 -8208.943} C_VEL
LIN {X 0,Y 453.432,Z 392.627,A -85,B 0,C 180,E1 -8211.839,E2 -8211.839} C_VEL
LIN {X 0,Y 453.52,Z 392.617,A -85,B 0,C 180,E1 -8214.735,E2 -8214.735} C_VEL
LIN {X 0,Y 453.539,Z 392.613,A -85,B 0,C 180,E1 -8217.96,E2 -8217.96} C_VEL
LIN {X 0,Y 453.471,Z 392.624,A -85,B 0,C 180,E1 -8221.525,E2 -8221.525} C_VEL
LIN {X 0,Y 453.488,Z 392.625,A -85,B 0,C 180,E1 -8224.777,E2 -8224.777} C_VEL
LIN {X 0,Y 453.468,Z 392.617,A -85,B 0,C 180,E1 -8228.312,E2 -8228.312} C_VEL
LIN {X 0,Y 453.499,Z 392.624,A -85,B 0,C 180,E1 -8230.609,E2 -8230.609} C_VEL
LIN {X 0,Y 453.461,Z 392.622,A -85,B 0,C 180,E1 -8233.244,E2 -8233.244} C_VEL
LIN {X 0,Y 453.479,Z 392.619,A -85,B 0,C 180,E1 -8235.78,E2 -8235.78} C_VEL
LIN {X 0,Y 453.487,Z 392.623,A -85,B 0,C 180,E1 -8238.21,E2 -8238.21} C_VEL
LIN {X 0,Y 453.5,Z 392.601,A -85,B 0,C 180,E1 -8240.793,E2 -8240.793} C_VEL
LIN {X 0,Y 453.462,Z 392.622,A -85,B 0,C 180,E1 -8243.917,E2 -8243.917} C_VEL
LIN {X 0,Y 453.488,Z 392.616,A -85,B 0,C 180,E1 -8247.151,E2 -8247.151} C_VEL
LIN {X 0,Y 453.478,Z 392.599,A -85,B 0,C 180,E1 -8250.268,E2 -8250.268} C_VEL
LIN {X 0,Y 453.506,Z 392.611,A -85,B 0,C 180,E1 -8253.294,E2 -8253.294} C_VEL
LIN {X 0,Y 453.502,Z 392.618,A -85,B 0,C 180,E1 -8256.238,E2 -8256.238} C_VEL
LIN {X 0,Y 453.486,Z 392.621,A -85,B 0,C 180,E1 -8259.118,E2 -8259.118} C_VEL
LIN {X 0,Y 453.508,Z 392.62,A -85,B 0,C 180,E1 -8261.944,E2 -8261.944} C_VEL
LIN {X 0,Y 453.518,Z 392.662,A -85,B 0,C 180,E1 -8262.953,E2 -8262.953} C_VEL
LIN {X 0,Y 457.76,Z 406.553,A -85,B 0,C 180,E1 -8263.869,E2 -8263.869} C_VEL
LIN {X 0,Y 457.202,Z 419.57,A -85,B 0,C 180,E1 -8264.737,E2 -8264.737} C_VEL
LIN {X 0,Y 456.576,Z 431.712,A -85,B 0,C 180,E1 -8265.742,E2 -8265.742} C_VEL
LIN {X 0,Y 455.913,Z 442.769,A -85,B 0,C 180,E1 -8266.857,E2 -8266.857} C_VEL
LIN {X 0,Y 455.279,Z 452.047,A -85,B 0,C 180,E1 -8267.971,E2 -8267.971} C_VEL
LIN {X 0,Y 454.732,Z 461.348,A -85,B 0,C 180,E1 -8269.312,E2 -8269.312} C_VEL
LIN {X 0,Y 454.321,Z 469.094,A -85,B 0,C 180,E1 -8270.652,E2 -8270.652} C_VEL
LIN {X 0,Y 453.858,Z 476.967,A -85,B 0,C 180,E1 -8272.327,E2 -8272.327} C_VEL
LIN {X 0,Y 453.612,Z 482.439,A -85,B 0,C 180,E1 -8273.774,E2 -8273.774} C_VEL
LIN {X 0,Y 453.337,Z 487.649,A -85,B 0,C 180,E1 -8275.554,E2 -8275.554} C_VEL
LIN {X 0,Y 453.13,Z 491.37,A -85,B 0,C 180,E1 -8277.333,E2 -8277.333} C_VEL
LIN {X 0,Y 453.08,Z 493.693,A -85,B 0,C 180,E1 -8279.111,E2 -8279.111} C_VEL
LIN {X 0,Y 453.079,Z 494.689,A -85,B 0,C 180,E1 -8280.889,E2 -8280.889} C_VEL
LIN {X 0,Y 453.211,Z 494.36,A -85,B 0,C 180,E1 -8282.666,E2 -8282.666} C_VEL
LIN {X 0,Y 453.287,Z 492.709,A -85,B 0,C 180,E1 -8284.446,E2 -8284.446} C_VEL
LIN {X 0,Y 453.601,Z 489.644,A -85,B 0,C 180,E1 -8286.226,E2 -8286.226} C_VEL
LIN {X 0,Y 453.814,Z 485.135,A -85,B 0,C 180,E1 -8288.012,E2 -8288.012} C_VEL
LIN {X 0,Y 454.189,Z 479.006,A -85,B 0,C 180,E1 -8289.8,E2 -8289.8} C_VEL
LIN {X 0,Y 454.671,Z 472.092,A -85,B 0,C 180,E1 -8291.366,E2 -8291.366} C_VEL
LIN {X 0,Y 455.299,Z 463.472,A -85,B 0,C 180,E1 -8292.923,E2 -8292.923} C_VEL
LIN {X 0,Y 455.936,Z 454.319,A -85,B 0,C 180,E1 -8294.278,E2 -8294.278} C_VEL
LIN {X 0,Y 456.628,Z 443.219,A -85,B 0,C 180,E1 -8295.625,E2 -8295.625} C_VEL
LIN {X 0,Y 457.355,Z 431.868,A -85,B 0,C 180,E1 -8296.746,E2 -8296.746} C_VEL
LIN {X 0,Y 457.99,Z 420.074,A -85,B 0,C 180,E1 -8297.696,E2 -8297.696} C_VEL
LIN {X 0,Y 458.551,Z 408.819,A -85,B 0,C 180,E1 -8298.427,E2 -8298.427} C_VEL
LIN {X 0,Y 458.012,Z 405.741,A -85,B 0,C 180,E1 -8298.635,E2 -8298.635} C_VEL
LIN {X 0,Y 454.465,Z 395.309,A -85,B 0,C 180,E1 -8299.381,E2 -8299.381} C_VEL
LIN {X 0,Y 453.551,Z 392.617,A -85,B 0,C 180,E1 -8299.584,E2 -8299.584} C_VEL
LIN {X 0,Y 453.483,Z 392.629,A -85,B 0,C 180,E1 -8302.795,E2 -8302.795} C_VEL
LIN {X 0,Y 453.521,Z 392.62,A -85,B 0,C 180,E1 -8305.998,E2 -8305.998} C_VEL
LIN {X 0,Y 453.513,Z 392.618,A -85,B 0,C 180,E1 -8308.711,E2 -8308.711} C_VEL
LIN {X 0,Y 453.467,Z 392.625,A -85,B 0,C 180,E1 -8311.799,E2 -8311.799} C_VEL
LIN {X 0,Y 453.483,Z 392.624,A -85,B 0,C 180,E1 -8314.989,E2 -8314.989} C_VEL
LIN {X 0,Y 453.467,Z 392.627,A -85,B 0,C 180,E1 -8318.311,E2 -8318.311} C_VEL
LIN {X 0,Y 453.497,Z 392.623,A -85,B 0,C 180,E1 -8320.609,E2 -8320.609} C_VEL
LIN {X 0,Y 453.459,Z 392.627,A -85,B 0,C 180,E1 -8323.244,E2 -8323.244} C_VEL
LIN {X 0,Y 453.458,Z 392.632,A -85,B 0,C 180,E1 -8326.305,E2 -8326.305} C_VEL
LIN {X 0,Y 453.487,Z 392.791,A -85,B 0,C 180,E1 -8326.752,E2 -8326.752} C_VEL
LIN {X 0,Y 454.812,Z 399.061,A -85,B 0,C 180,E1 -8329.216,E2 -8329.216} C_VEL
LIN {X 0,Y 455.584,Z 403.573,A -85,B 0,C 180,E1 -8330.766,E2 -8330.766} C_VEL
LIN {X 0,Y 455.523,Z 407.25,A -85,B 0,C 180,E1 -8331.892,E2 -8331.892} C_VEL
LIN {X 0,Y 454.485,Z 420.834,A -85,B 0,C 180,E1 -8335.637,E2 -8335.637} C_VEL
LIN {X 0,Y 454.238,Z 431.3,A -85,B 0,C 180,E1 -8338.317,E2 -8338.317} C_VEL
LIN {X 0,Y 453.995,Z 443.666,A -85,B 0,C 180,E1 -8341.321,E2 -8341.321} C_VEL
LIN {X 0,Y 453.757,Z 458.526,A -85,B 0,C 180,E1 -8344.79,E2 -8344.79} C_VEL
LIN {X 0,Y 453.532,Z 473.422,A -85,B 0,C 180,E1 -8348.166,E2 -8348.166} C_VEL
LIN {X 0,Y 453.376,Z 484.707,A -85,B 0,C 180,E1 -8350.69,E2 -8350.69} C_VEL
LIN {X 0,Y 455.313,Z 501.559,A -85,B 0,C 180,E1 -8351.217,E2 -8351.217} C_VEL
LIN {X 0,Y 456.33,Z 515.169,A -85,B 0,C 180,E1 -8351.769,E2 -8351.769} C_VEL
LIN {X 0,Y 457.095,Z 521.581,A -85,B 0,C 180,E1 -8352.09,E2 -8352.09} C_VEL
LIN {X 0,Y 456.381,Z 535.327,A -85,B 0,C 180,E1 -8352.821,E2 -8352.821} C_VEL
LIN {X 0,Y 455.596,Z 549.295,A -85,B 0,C 180,E1 -8353.763,E2 -8353.763} C_VEL
LIN {X 0,Y 454.819,Z 562.698,A -85,B 0,C 180,E1 -8354.884,E2 -8354.884} C_VEL
LIN {X 0,Y 454.204,Z 574.846,A -85,B 0,C 180,E1 -8356.122,E2 -8356.122} C_VEL
LIN {X 0,Y 453.692,Z 585.81,A -85,B 0,C 180,E1 -8357.474,E2 -8357.474} C_VEL
LIN {X 0,Y 453.371,Z 594.927,A -85,B 0,C 180,E1 -8358.826,E2 -8358.826} C_VEL
LIN {X 0,Y 453.104,Z 603.679,A -85,B 0,C 180,E1 -8360.401,E2 -8360.401} C_VEL
LIN {X 0,Y 452.954,Z 610.761,A -85,B 0,C 180,E1 -8361.972,E2 -8361.972} C_VEL
LIN {X 0,Y 452.888,Z 617.076,A -85,B 0,C 180,E1 -8363.763,E2 -8363.763} C_VEL
LIN {X 0,Y 452.946,Z 620.713,A -85,B 0,C 180,E1 -8365.104,E2 -8365.104} C_VEL
LIN {X 0,Y 452.899,Z 623.43,A -85,B 0,C 180,E1 -8366.44,E2 -8366.44} C_VEL
LIN {X 0,Y 452.853,Z 625.745,A -85,B 0,C 180,E1 -8368.22,E2 -8368.22} C_VEL
LIN {X 0,Y 452.948,Z 626.616,A -85,B 0,C 180,E1 -8369.999,E2 -8369.999} C_VEL
LIN {X 0,Y 452.817,Z 626.01,A -85,B 0,C 180,E1 -8371.778,E2 -8371.778} C_VEL
LIN {X 0,Y 452.836,Z 623.987,A -85,B 0,C 180,E1 -8373.558,E2 -8373.558} C_VEL
LIN {X 0,Y 452.804,Z 620.473,A -85,B 0,C 180,E1 -8375.342,E2 -8375.342} C_VEL
LIN {X 0,Y 452.842,Z 616.943,A -85,B 0,C 180,E1 -8376.653,E2 -8376.653} C_VEL
LIN {X 0,Y 452.843,Z 612.204,A -85,B 0,C 180,E1 -8378.028,E2 -8378.028} C_VEL
LIN {X 0,Y 453.028,Z 605.506,A -85,B 0,C 180,E1 -8379.599,E2 -8379.599} C_VEL
LIN {X 0,Y 453.343,Z 597.19,A -85,B 0,C 180,E1 -8381.173,E2 -8381.173} C_VEL
LIN {X 0,Y 453.718,Z 587.822,A -85,B 0,C 180,E1 -8382.615,E2 -8382.615} C_VEL
LIN {X 0,Y 454.263,Z 577.991,A -85,B 0,C 180,E1 -8383.874,E2 -8383.874} C_VEL
LIN {X 0,Y 454.909,Z 566.316,A -85,B 0,C 180,E1 -8385.111,E2 -8385.111} C_VEL
LIN {X 0,Y 455.688,Z 554.768,A -85,B 0,C 180,E1 -8386.116,E2 -8386.116} C_VEL
LIN {X 0,Y 456.41,Z 542.218,A -85,B 0,C 180,E1 -8387.011,E2 -8387.011} C_VEL
LIN {X 0,Y 457.078,Z 529.094,A -85,B 0,C 180,E1 -8387.754,E2 -8387.754} C_VEL
LIN {X 0,Y 457.479,Z 521.066,A -85,B 0,C 180,E1 -8388.124,E2 -8388.124} C_VEL
LIN {X 0,Y 455.723,Z 506.969,A -85,B 0,C 180,E1 -8388.705,E2 -8388.705} C_VEL
LIN {X 0,Y 453.531,Z 491.169,A -85,B 0,C 180,E1 -8389.18,E2 -8389.18} C_VEL
LIN {X 0,Y 453.963,Z 476.34,A -85,B 0,C 180,E1 -8392.769,E2 -8392.769} C_VEL
LIN {X 0,Y 454.519,Z 462.196,A -85,B 0,C 180,E1 -8396.256,E2 -8396.256} C_VEL
LIN {X 0,Y 455.258,Z 446.68,A -85,B 0,C 180,E1 -8400.175,E2 -8400.175} C_VEL
LIN {X 0,Y 455.957,Z 433.104,A -85,B 0,C 180,E1 -8403.702,E2 -8403.702} C_VEL
LIN {X 0,Y 456.815,Z 419.22,A -85,B 0,C 180,E1 -8407.422,E2 -8407.422} C_VEL
LIN {X 0,Y 457.229,Z 412.04,A -85,B 0,C 180,E1 -8409.409,E2 -8409.409} C_VEL
LIN {X 0,Y 456.143,Z 405.074,A -85,B 0,C 180,E1 -8411.49,E2 -8411.49} C_VEL
LIN {X 0,Y 453.714,Z 393.776,A -85,B 0,C 180,E1 -8415.068,E2 -8415.068} C_VEL
LIN {X 0,Y 453.486,Z 392.623,A -85,B 0,C 180,E1 -8415.469,E2 -8415.469} C_VEL
LIN {X 0,Y 453.489,Z 392.622,A -85,B 0,C 180,E1 -8418.211,E2 -8418.211} C_VEL
LIN {X 0,Y 453.527,Z 392.615,A -85,B 0,C 180,E1 -8420.786,E2 -8420.786} C_VEL
LIN {X 0,Y 453.449,Z 392.626,A -85,B 0,C 180,E1 -8423.917,E2 -8423.917} C_VEL
LIN {X 0,Y 453.474,Z 392.624,A -85,B 0,C 180,E1 -8427.151,E2 -8427.151} C_VEL
LIN {X 0,Y 453.504,Z 392.618,A -85,B 0,C 180,E1 -8430.271,E2 -8430.271} C_VEL
LIN {X 0,Y 453.504,Z 392.622,A -85,B 0,C 180,E1 -8433.294,E2 -8433.294} C_VEL
LIN {X 0,Y 453.493,Z 392.62,A -85,B 0,C 180,E1 -8436.238,E2 -8436.238} C_VEL
LIN {X 0,Y 453.473,Z 392.624,A -85,B 0,C 180,E1 -8439.117,E2 -8439.117} C_VEL
LIN {X 0,Y 453.501,Z 392.619,A -85,B 0,C 180,E1 -8441.944,E2 -8441.944} C_VEL
LIN {X 0,Y 453.53,Z 392.615,A -85,B 0,C 180,E1 -8444.726,E2 -8444.726} C_VEL
LIN {X 0,Y 453.591,Z 392.61,A -85,B 0,C 180,E1 -8447.472,E2 -8447.472} C_VEL
LIN {X 0,Y 453.583,Z 392.611,A -85,B 0,C 180,E1 -8451.087,E2 -8451.087} C_VEL
LIN {X 0,Y 453.667,Z 392.598,A -85,B 0,C 180,E1 -8453.775,E2 -8453.775} C_VEL
LIN {X 0,Y 453.756,Z 392.59,A -85,B 0,C 180,E1 -8457.337,E2 -8457.337} C_VEL
LIN {X 0,Y 453.814,Z 392.58,A -85,B 0,C 180,E1 -8460,E2 -8460} C_VEL
LIN {X 0,Y 453.756,Z 392.587,A -85,B 0,C 180,E1 -8462.663,E2 -8462.663} C_VEL
LIN {X 0,Y 453.67,Z 392.598,A -85,B 0,C 180,E1 -8466.226,E2 -8466.226} C_VEL
LIN {X 0,Y 453.583,Z 392.611,A -85,B 0,C 180,E1 -8468.914,E2 -8468.914} C_VEL
LIN {X 0,Y 453.591,Z 392.608,A -85,B 0,C 180,E1 -8472.551,E2 -8472.551} C_VEL
LIN {X 0,Y 453.534,Z 392.615,A -85,B 0,C 180,E1 -8476.197,E2 -8476.197} C_VEL
LIN {X 0,Y 453.511,Z 392.622,A -85,B 0,C 180,E1 -8479.042,E2 -8479.042} C_VEL
LIN {X 0,Y 453.467,Z 392.623,A -85,B 0,C 180,E1 -8481.837,E2 -8481.837} C_VEL
LIN {X 0,Y 453.506,Z 392.62,A -85,B 0,C 180,E1 -8484.735,E2 -8484.735} C_VEL
LIN {X 0,Y 453.529,Z 392.616,A -85,B 0,C 180,E1 -8487.962,E2 -8487.962} C_VEL
LIN {X 0,Y 453.459,Z 392.624,A -85,B 0,C 180,E1 -8491.526,E2 -8491.526} C_VEL
LIN {X 0,Y 453.482,Z 392.624,A -85,B 0,C 180,E1 -8494.779,E2 -8494.779} C_VEL
LIN {X 0,Y 453.467,Z 392.623,A -85,B 0,C 180,E1 -8498.312,E2 -8498.312} C_VEL
LIN {X 0,Y 453.488,Z 392.622,A -85,B 0,C 180,E1 -8500.61,E2 -8500.61} C_VEL
LIN {X 0,Y 453.471,Z 392.623,A -85,B 0,C 180,E1 -8504.221,E2 -8504.221} C_VEL
LIN {X 0,Y 453.459,Z 392.626,A -85,B 0,C 180,E1 -8507.006,E2 -8507.006} C_VEL
LIN {X 0,Y 453.53,Z 392.617,A -85,B 0,C 180,E1 -8510.556,E2 -8510.556} C_VEL
LIN {X 0,Y 453.455,Z 392.625,A -85,B 0,C 180,E1 -8513.919,E2 -8513.919} C_VEL
LIN {X 0,Y 453.481,Z 392.622,A -85,B 0,C 180,E1 -8517.153,E2 -8517.153} C_VEL
LIN {X 0,Y 453.474,Z 392.623,A -85,B 0,C 180,E1 -8520.27,E2 -8520.27} C_VEL
LIN {X 0,Y 453.509,Z 392.618,A -85,B 0,C 180,E1 -8523.296,E2 -8523.296} C_VEL
LIN {X 0,Y 453.503,Z 392.619,A -85,B 0,C 180,E1 -8526.24,E2 -8526.24} C_VEL
LIN {X 0,Y 453.483,Z 392.621,A -85,B 0,C 180,E1 -8529.119,E2 -8529.119} C_VEL
LIN {X 0,Y 453.511,Z 392.618,A -85,B 0,C 180,E1 -8531.946,E2 -8531.946} C_VEL
LIN {X 0,Y 453.491,Z 392.623,A -85,B 0,C 180,E1 -8534.726,E2 -8534.726} C_VEL
LIN {X 0,Y 453.329,Z 392.809,A -85,B 0,C 180,E1 -8537.293,E2 -8537.293} C_VEL
LIN {X 0,Y 457.042,Z 405.063,A -85,B 0,C 180,E1 -8537.786,E2 -8537.786} C_VEL
LIN {X 0,Y 456.839,Z 416.725,A -85,B 0,C 180,E1 -8538.287,E2 -8538.287} C_VEL
LIN {X 0,Y 456.712,Z 421.473,A -85,B 0,C 180,E1 -8538.539,E2 -8538.539} C_VEL
LIN {X 0,Y 455.929,Z 426.846,A -85,B 0,C 180,E1 -8538.837,E2 -8538.837} C_VEL
LIN {X 0,Y 451.433,Z 438.767,A -85,B 0,C 180,E1 -8539.543,E2 -8539.543} C_VEL
LIN {X 0,Y 449.262,Z 445.279,A -85,B 0,C 180,E1 -8540.042,E2 -8540.042} C_VEL
LIN {X 0,Y 448.824,Z 448.411,A -85,B 0,C 180,E1 -8540.337,E2 -8540.337} C_VEL
LIN {X 0,Y 448.308,Z 458.198,A -85,B 0,C 180,E1 -8541.433,E2 -8541.433} C_VEL
LIN {X 0,Y 447.865,Z 466.406,A -85,B 0,C 180,E1 -8542.563,E2 -8542.563} C_VEL
LIN {X 0,Y 447.392,Z 474.352,A -85,B 0,C 180,E1 -8543.914,E2 -8543.914} C_VEL
LIN {X 0,Y 447.014,Z 479.801,A -85,B 0,C 180,E1 -8545.04,E2 -8545.04} C_VEL
LIN {X 0,Y 446.733,Z 485.094,A -85,B 0,C 180,E1 -8546.393,E2 -8546.393} C_VEL
LIN {X 0,Y 446.552,Z 489.23,A -85,B 0,C 180,E1 -8547.746,E2 -8547.746} C_VEL
LIN {X 0,Y 446.313,Z 492.352,A -85,B 0,C 180,E1 -8549.099,E2 -8549.099} C_VEL
LIN {X 0,Y 446.226,Z 493.898,A -85,B 0,C 180,E1 -8550.001,E2 -8550.001} C_VEL
LIN {X 0,Y 446.091,Z 495.07,A -85,B 0,C 180,E1 -8550.904,E2 -8550.904} C_VEL
LIN {X 0,Y 446.158,Z 495.79,A -85,B 0,C 180,E1 -8551.806,E2 -8551.806} C_VEL
LIN {X 0,Y 446.096,Z 496.132,A -85,B 0,C 180,E1 -8553.614,E2 -8553.614} C_VEL
LIN {X 0,Y 446.161,Z 495.733,A -85,B 0,C 180,E1 -8554.518,E2 -8554.518} C_VEL
LIN {X 0,Y 446.308,Z 494.899,A -85,B 0,C 180,E1 -8555.422,E2 -8555.422} C_VEL
LIN {X 0,Y 446.412,Z 492.109,A -85,B 0,C 180,E1 -8557.236,E2 -8557.236} C_VEL
LIN {X 0,Y 446.603,Z 488.879,A -85,B 0,C 180,E1 -8558.599,E2 -8558.599} C_VEL
LIN {X 0,Y 446.958,Z 484.578,A -85,B 0,C 180,E1 -8559.961,E2 -8559.961} C_VEL
LIN {X 0,Y 447.331,Z 478.022,A -85,B 0,C 180,E1 -8561.556,E2 -8561.556} C_VEL
LIN {X 0,Y 447.706,Z 470.992,A -85,B 0,C 180,E1 -8562.906,E2 -8562.906} C_VEL
LIN {X 0,Y 448.251,Z 463.531,A -85,B 0,C 180,E1 -8564.066,E2 -8564.066} C_VEL
LIN {X 0,Y 448.738,Z 454.606,A -85,B 0,C 180,E1 -8565.209,E2 -8565.209} C_VEL
LIN {X 0,Y 449.25,Z 444.666,A -85,B 0,C 180,E1 -8566.239,E2 -8566.239} C_VEL
LIN {X 0,Y 449.779,Z 433.65,A -85,B 0,C 180,E1 -8567.154,E2 -8567.154} C_VEL
LIN {X 0,Y 450.219,Z 421.844,A -85,B 0,C 180,E1 -8567.918,E2 -8567.918} C_VEL
LIN {X 0,Y 450.507,Z 408.943,A -85,B 0,C 180,E1 -8568.534,E2 -8568.534} C_VEL
LIN {X 0,Y 450.228,Z 405.773,A -85,B 0,C 180,E1 -8568.67,E2 -8568.67} C_VEL
LIN {X 0,Y 446.23,Z 393.528,A -85,B 0,C 180,E1 -8569.219,E2 -8569.219} C_VEL
LIN {X 0,Y 446.391,Z 393.504,A -85,B 0,C 180,E1 -8572.202,E2 -8572.202} C_VEL
LIN {X 0,Y 446.464,Z 393.495,A -85,B 0,C 180,E1 -8575.153,E2 -8575.153} C_VEL
LIN {X 0,Y 446.491,Z 393.491,A -85,B 0,C 180,E1 -8578.179,E2 -8578.179} C_VEL
LIN {X 0,Y 446.424,Z 393.501,A -85,B 0,C 180,E1 -8581.775,E2 -8581.775} C_VEL
LIN {X 0,Y 446.429,Z 393.504,A -85,B 0,C 180,E1 -8584.524,E2 -8584.524} C_VEL
LIN {X 0,Y 446.42,Z 393.495,A -85,B 0,C 180,E1 -8588.079,E2 -8588.079} C_VEL
LIN {X 0,Y 446.432,Z 393.5,A -85,B 0,C 180,E1 -8590.918,E2 -8590.918} C_VEL
LIN {X 0,Y 446.407,Z 393.502,A -85,B 0,C 180,E1 -8593.846,E2 -8593.846} C_VEL
LIN {X 0,Y 446.426,Z 393.502,A -85,B 0,C 180,E1 -8596.4,E2 -8596.4} C_VEL
LIN {X 0,Y 446.449,Z 393.493,A -85,B 0,C 180,E1 -8599.802,E2 -8599.802} C_VEL
LIN {X 0,Y 446.433,Z 393.486,A -85,B 0,C 180,E1 -8602.123,E2 -8602.123} C_VEL
LIN {X 0,Y 446.435,Z 393.499,A -85,B 0,C 180,E1 -8605.477,E2 -8605.477} C_VEL
LIN {X 0,Y 446.42,Z 393.486,A -85,B 0,C 180,E1 -8608.7,E2 -8608.7} C_VEL
LIN {X 0,Y 446.489,Z 393.476,A -85,B 0,C 180,E1 -8611.821,E2 -8611.821} C_VEL
LIN {X 0,Y 446.448,Z 393.495,A -85,B 0,C 180,E1 -8614.847,E2 -8614.847} C_VEL
LIN {X 0,Y 446.452,Z 393.496,A -85,B 0,C 180,E1 -8618.245,E2 -8618.245} C_VEL
LIN {X 0,Y 446.456,Z 393.5,A -85,B 0,C 180,E1 -8621.649,E2 -8621.649} C_VEL
LIN {X 0,Y 446.464,Z 393.496,A -85,B 0,C 180,E1 -8622.681,E2 -8622.681} C_VEL
LIN {X 0,Y 450.745,Z 407.475,A -85,B 0,C 180,E1 -8623.638,E2 -8623.638} C_VEL
LIN {X 0,Y 450.574,Z 415.446,A -85,B 0,C 180,E1 -8624.159,E2 -8624.159} C_VEL
LIN {X 0,Y 449.895,Z 428.498,A -85,B 0,C 180,E1 -8625.179,E2 -8625.179} C_VEL
LIN {X 0,Y 449.269,Z 439.635,A -85,B 0,C 180,E1 -8626.243,E2 -8626.243} C_VEL
LIN {X 0,Y 448.591,Z 449.213,A -85,B 0,C 180,E1 -8627.33,E2 -8627.33} C_VEL
LIN {X 0,Y 447.956,Z 459.174,A -85,B 0,C 180,E1 -8628.69,E2 -8628.69} C_VEL
LIN {X 0,Y 447.476,Z 468.684,A -85,B 0,C 180,E1 -8630.279,E2 -8630.279} C_VEL
LIN {X 0,Y 446.995,Z 476.406,A -85,B 0,C 180,E1 -8631.865,E2 -8631.865} C_VEL
LIN {X 0,Y 446.725,Z 481.767,A -85,B 0,C 180,E1 -8633.224,E2 -8633.224} C_VEL
LIN {X 0,Y 446.442,Z 487.456,A -85,B 0,C 180,E1 -8635.033,E2 -8635.033} C_VEL
LIN {X 0,Y 446.21,Z 490.662,A -85,B 0,C 180,E1 -8636.388,E2 -8636.388} C_VEL
LIN {X 0,Y 446.148,Z 493.696,A -85,B 0,C 180,E1 -8638.194,E2 -8638.194} C_VEL
LIN {X 0,Y 446.056,Z 495.397,A -85,B 0,C 180,E1 -8640,E2 -8640} C_VEL
LIN {X 0,Y 446.15,Z 495.755,A -85,B 0,C 180,E1 -8641.805,E2 -8641.805} C_VEL
LIN {X 0,Y 446.202,Z 494.8,A -85,B 0,C 180,E1 -8643.612,E2 -8643.612} C_VEL
LIN {X 0,Y 446.401,Z 492.462,A -85,B 0,C 180,E1 -8645.42,E2 -8645.42} C_VEL
LIN {X 0,Y 446.653,Z 489.783,A -85,B 0,C 180,E1 -8646.777,E2 -8646.777} C_VEL
LIN {X 0,Y 446.89,Z 486.247,A -85,B 0,C 180,E1 -8648.137,E2 -8648.137} C_VEL
LIN {X 0,Y 447.302,Z 480.135,A -85,B 0,C 180,E1 -8649.952,E2 -8649.952} C_VEL
LIN {X 0,Y 447.803,Z 473.266,A -85,B 0,C 180,E1 -8651.543,E2 -8651.543} C_VEL
LIN {X 0,Y 448.508,Z 464.66,A -85,B 0,C 180,E1 -8653.126,E2 -8653.126} C_VEL
LIN {X 0,Y 449.187,Z 455.537,A -85,B 0,C 180,E1 -8654.497,E2 -8654.497} C_VEL
LIN {X 0,Y 449.9,Z 444.455,A -85,B 0,C 180,E1 -8655.865,E2 -8655.865} C_VEL
LIN {X 0,Y 450.668,Z 433.144,A -85,B 0,C 180,E1 -8657.001,E2 -8657.001} C_VEL
LIN {X 0,Y 451.376,Z 421.277,A -85,B 0,C 180,E1 -8657.978,E2 -8657.978} C_VEL
LIN {X 0,Y 451.968,Z 410.364,A -85,B 0,C 180,E1 -8658.706,E2 -8658.706} C_VEL
LIN {X 0,Y 450.496,Z 404.808,A -85,B 0,C 180,E1 -8659.124,E2 -8659.124} C_VEL
LIN {X 0,Y 446.479,Z 393.498,A -85,B 0,C 180,E1 -8659.935,E2 -8659.935} C_VEL
LIN {X 0,Y 446.433,Z 393.506,A -85,B 0,C 180,E1 -8663.176,E2 -8663.176} C_VEL
LIN {X 0,Y 446.478,Z 393.498,A -85,B 0,C 180,E1 -8666.202,E2 -8666.202} C_VEL
LIN {X 0,Y 446.451,Z 393.501,A -85,B 0,C 180,E1 -8669.209,E2 -8669.209} C_VEL
LIN {X 0,Y 446.425,Z 393.502,A -85,B 0,C 180,E1 -8672.361,E2 -8672.361} C_VEL
LIN {X 0,Y 446.422,Z 393.505,A -85,B 0,C 180,E1 -8675.626,E2 -8675.626} C_VEL
LIN {X 0,Y 446.447,Z 393.501,A -85,B 0,C 180,E1 -8679.027,E2 -8679.027} C_VEL
LIN {X 0,Y 446.437,Z 393.502,A -85,B 0,C 180,E1 -8682.277,E2 -8682.277} C_VEL
LIN {X 0,Y 446.456,Z 393.502,A -85,B 0,C 180,E1 -8685.103,E2 -8685.103} C_VEL
LIN {X 0,Y 446.452,Z 393.717,A -85,B 0,C 180,E1 -8686.276,E2 -8686.276} C_VEL
LIN {X 0,Y 447.789,Z 400.047,A -85,B 0,C 180,E1 -8688.882,E2 -8688.882} C_VEL
LIN {X 0,Y 448.701,Z 405.164,A -85,B 0,C 180,E1 -8690.701,E2 -8690.701} C_VEL
LIN {X 0,Y 448.372,Z 410.404,A -85,B 0,C 180,E1 -8692.315,E2 -8692.315} C_VEL
LIN {X 0,Y 447.458,Z 423.64,A -85,B 0,C 180,E1 -8696.013,E2 -8696.013} C_VEL
LIN {X 0,Y 447.106,Z 436.292,A -85,B 0,C 180,E1 -8699.278,E2 -8699.278} C_VEL
LIN {X 0,Y 446.849,Z 446.752,A -85,B 0,C 180,E1 -8701.846,E2 -8701.846} C_VEL
LIN {X 0,Y 446.683,Z 459.452,A -85,B 0,C 180,E1 -8704.861,E2 -8704.861} C_VEL
LIN {X 0,Y 446.425,Z 474.116,A -85,B 0,C 180,E1 -8708.253,E2 -8708.253} C_VEL
LIN {X 0,Y 446.356,Z 483.122,A -85,B 0,C 180,E1 -8710.304,E2 -8710.304} C_VEL
LIN {X 0,Y 448.469,Z 501.206,A -85,B 0,C 180,E1 -8710.92,E2 -8710.92} C_VEL
LIN {X 0,Y 449.406,Z 515.099,A -85,B 0,C 180,E1 -8711.512,E2 -8711.512} C_VEL
LIN {X 0,Y 450.232,Z 521.813,A -85,B 0,C 180,E1 -8711.867,E2 -8711.867} C_VEL
LIN {X 0,Y 449.457,Z 535.681,A -85,B 0,C 180,E1 -8712.644,E2 -8712.644} C_VEL
LIN {X 0,Y 448.685,Z 548.103,A -85,B 0,C 180,E1 -8713.506,E2 -8713.506} C_VEL
LIN {X 0,Y 447.899,Z 561.469,A -85,B 0,C 180,E1 -8714.645,E2 -8714.645} C_VEL
LIN {X 0,Y 447.177,Z 573.601,A -85,B 0,C 180,E1 -8715.9,E2 -8715.9} C_VEL
LIN {X 0,Y 446.663,Z 584.764,A -85,B 0,C 180,E1 -8717.3,E2 -8717.3} C_VEL
LIN {X 0,Y 446.307,Z 593.713,A -85,B 0,C 180,E1 -8718.647,E2 -8718.647} C_VEL
LIN {X 0,Y 446.026,Z 602.493,A -85,B 0,C 180,E1 -8720.247,E2 -8720.247} C_VEL
LIN {X 0,Y 445.882,Z 609.607,A -85,B 0,C 180,E1 -8721.844,E2 -8721.844} C_VEL
LIN {X 0,Y 445.843,Z 614.74,A -85,B 0,C 180,E1 -8723.263,E2 -8723.263} C_VEL
LIN {X 0,Y 445.901,Z 619.626,A -85,B 0,C 180,E1 -8725.026,E2 -8725.026} C_VEL
LIN {X 0,Y 445.865,Z 622.368,A -85,B 0,C 180,E1 -8726.384,E2 -8726.384} C_VEL
LIN {X 0,Y 445.822,Z 624.709,A -85,B 0,C 180,E1 -8728.192,E2 -8728.192} C_VEL
LIN {X 0,Y 445.932,Z 625.601,A -85,B 0,C 180,E1 -8729.999,E2 -8729.999} C_VEL
LIN {X 0,Y 445.783,Z 625.003,A -85,B 0,C 180,E1 -8731.806,E2 -8731.806} C_VEL
LIN {X 0,Y 445.796,Z 622.984,A -85,B 0,C 180,E1 -8733.614,E2 -8733.614} C_VEL
LIN {X 0,Y 445.745,Z 619.467,A -85,B 0,C 180,E1 -8735.427,E2 -8735.427} C_VEL
LIN {X 0,Y 445.771,Z 616.225,A -85,B 0,C 180,E1 -8736.659,E2 -8736.659} C_VEL
LIN {X 0,Y 445.793,Z 611.188,A -85,B 0,C 180,E1 -8738.156,E2 -8738.156} C_VEL
LIN {X 0,Y 445.937,Z 604.464,A -85,B 0,C 180,E1 -8739.753,E2 -8739.753} C_VEL
LIN {X 0,Y 446.282,Z 596.116,A -85,B 0,C 180,E1 -8741.352,E2 -8741.352} C_VEL
LIN {X 0,Y 446.667,Z 587.383,A -85,B 0,C 180,E1 -8742.724,E2 -8742.724} C_VEL
LIN {X 0,Y 447.275,Z 576.844,A -85,B 0,C 180,E1 -8744.095,E2 -8744.095} C_VEL
LIN {X 0,Y 447.969,Z 565.123,A -85,B 0,C 180,E1 -8745.351,E2 -8745.351} C_VEL
LIN {X 0,Y 448.765,Z 553.52,A -85,B 0,C 180,E1 -8746.372,E2 -8746.372} C_VEL
LIN {X 0,Y 449.561,Z 540.915,A -85,B 0,C 180,E1 -8747.278,E2 -8747.278} C_VEL
LIN {X 0,Y 450.256,Z 528.175,A -85,B 0,C 180,E1 -8748.008,E2 -8748.008} C_VEL
LIN {X 0,Y 450.465,Z 521.103,A -85,B 0,C 180,E1 -8748.346,E2 -8748.346} C_VEL
LIN {X 0,Y 448.848,Z 507.513,A -85,B 0,C 180,E1 -8748.933,E2 -8748.933} C_VEL
LIN {X 0,Y 446.707,Z 492.384,A -85,B 0,C 180,E1 -8749.415,E2 -8749.415} C_VEL
LIN {X 0,Y 446.46,Z 490.301,A -85,B 0,C 180,E1 -8749.489,E2 -8749.489} C_VEL
LIN {X 0,Y 446.88,Z 477.425,A -85,B 0,C 180,E1 -8752.661,E2 -8752.661} C_VEL
LIN {X 0,Y 447.434,Z 463.757,A -85,B 0,C 180,E1 -8756.09,E2 -8756.09} C_VEL
LIN {X 0,Y 448.036,Z 450.004,A -85,B 0,C 180,E1 -8759.61,E2 -8759.61} C_VEL
LIN {X 0,Y 448.603,Z 440.047,A -85,B 0,C 180,E1 -8762.222,E2 -8762.222} C_VEL
LIN {X 0,Y 449.14,Z 430.304,A -85,B 0,C 180,E1 -8764.828,E2 -8764.828} C_VEL
LIN {X 0,Y 450.031,Z 418.412,A -85,B 0,C 180,E1 -8768.085,E2 -8768.085} C_VEL
LIN {X 0,Y 450.299,Z 413.431,A -85,B 0,C 180,E1 -8769.492,E2 -8769.492} C_VEL
LIN {X 0,Y 449.353,Z 407.301,A -85,B 0,C 180,E1 -8771.346,E2 -8771.346} C_VEL
LIN {X 0,Y 446.895,Z 395.761,A -85,B 0,C 180,E1 -8775.045,E2 -8775.045} C_VEL
LIN {X 0,Y 446.434,Z 393.501,A -85,B 0,C 180,E1 -8775.867,E2 -8775.867} C_VEL
LIN {X 0,Y 446.44,Z 393.5,A -85,B 0,C 180,E1 -8779.078,E2 -8779.078} C_VEL
LIN {X 0,Y 446.431,Z 393.503,A -85,B 0,C 180,E1 -8781.916,E2 -8781.916} C_VEL
LIN {X 0,Y 446.422,Z 393.504,A -85,B 0,C 180,E1 -8785.476,E2 -8785.476} C_VEL
LIN {X 0,Y 446.41,Z 393.502,A -85,B 0,C 180,E1 -8788.699,E2 -8788.699} C_VEL
LIN {X 0,Y 446.474,Z 393.494,A -85,B 0,C 180,E1 -8791.821,E2 -8791.821} C_VEL
LIN {X 0,Y 446.448,Z 393.498,A -85,B 0,C 180,E1 -8794.847,E2 -8794.847} C_VEL
LIN {X 0,Y 446.437,Z 393.499,A -85,B 0,C 180,E1 -8798.245,E2 -8798.245} C_VEL
LIN {X 0,Y 446.447,Z 393.498,A -85,B 0,C 180,E1 -8801.649,E2 -8801.649} C_VEL
LIN {X 0,Y 446.498,Z 393.491,A -85,B 0,C 180,E1 -8804.48,E2 -8804.48} C_VEL
LIN {X 0,Y 446.529,Z 393.487,A -85,B 0,C 180,E1 -8808.194,E2 -8808.194} C_VEL
LIN {X 0,Y 446.589,Z 393.479,A -85,B 0,C 180,E1 -8811.858,E2 -8811.858} C_VEL
LIN {X 0,Y 446.636,Z 393.474,A -85,B 0,C 180,E1 -8814.583,E2 -8814.583} C_VEL
LIN {X 0,Y 446.7,Z 393.469,A -85,B 0,C 180,E1 -8817.295,E2 -8817.295} C_VEL
LIN {X 0,Y 446.784,Z 393.455,A -85,B 0,C 180,E1 -8820,E2 -8820} C_VEL
LIN {X 0,Y 446.7,Z 393.467,A -85,B 0,C 180,E1 -8822.706,E2 -8822.706} C_VEL
LIN {X 0,Y 446.638,Z 393.474,A -85,B 0,C 180,E1 -8826.324,E2 -8826.324} C_VEL
LIN {X 0,Y 446.529,Z 393.491,A -85,B 0,C 180,E1 -8829.056,E2 -8829.056} C_VEL
LIN {X 0,Y 446.524,Z 393.489,A -85,B 0,C 180,E1 -8832.73,E2 -8832.73} C_VEL
LIN {X 0,Y 446.48,Z 393.494,A -85,B 0,C 180,E1 -8836.46,E2 -8836.46} C_VEL
LIN {X 0,Y 446.46,Z 393.497,A -85,B 0,C 180,E1 -8839.304,E2 -8839.304} C_VEL
LIN {X 0,Y 446.409,Z 393.503,A -85,B 0,C 180,E1 -8842.2,E2 -8842.2} C_VEL
LIN {X 0,Y 446.45,Z 393.499,A -85,B 0,C 180,E1 -8845.153,E2 -8845.153} C_VEL
LIN {X 0,Y 446.476,Z 393.494,A -85,B 0,C 180,E1 -8848.18,E2 -8848.18} C_VEL
LIN {X 0,Y 446.412,Z 393.502,A -85,B 0,C 180,E1 -8851.776,E2 -8851.776} C_VEL
LIN {X 0,Y 446.423,Z 393.502,A -85,B 0,C 180,E1 -8854.524,E2 -8854.524} C_VEL
LIN {X 0,Y 446.424,Z 393.501,A -85,B 0,C 180,E1 -8858.083,E2 -8858.083} C_VEL
LIN {X 0,Y 446.422,Z 393.504,A -85,B 0,C 180,E1 -8860.919,E2 -8860.919} C_VEL
LIN {X 0,Y 446.42,Z 393.501,A -85,B 0,C 180,E1 -8863.844,E2 -8863.844} C_VEL
LIN {X 0,Y 446.395,Z 393.505,A -85,B 0,C 180,E1 -8866.405,E2 -8866.405} C_VEL
LIN {X 0,Y 446.465,Z 393.496,A -85,B 0,C 180,E1 -8869.806,E2 -8869.806} C_VEL
LIN {X 0,Y 446.431,Z 393.5,A -85,B 0,C 180,E1 -8872.125,E2 -8872.125} C_VEL
LIN {X 0,Y 446.428,Z 393.5,A -85,B 0,C 180,E1 -8875.479,E2 -8875.479} C_VEL
LIN {X 0,Y 446.416,Z 393.505,A -85,B 0,C 180,E1 -8878.701,E2 -8878.701} C_VEL
LIN {X 0,Y 446.484,Z 393.494,A -85,B 0,C 180,E1 -8881.823,E2 -8881.823} C_VEL
LIN {X 0,Y 446.458,Z 393.498,A -85,B 0,C 180,E1 -8884.849,E2 -8884.849} C_VEL
LIN {X 0,Y 446.449,Z 393.498,A -85,B 0,C 180,E1 -8888.246,E2 -8888.246} C_VEL
LIN {X 0,Y 446.457,Z 393.497,A -85,B 0,C 180,E1 -8891.65,E2 -8891.65} C_VEL
LIN {X 0,Y 446.449,Z 393.5,A -85,B 0,C 180,E1 -8894.479,E2 -8894.479} C_VEL
LIN {X 0,Y 446.291,Z 393.522,A -85,B 0,C 180,E1 -8897.042,E2 -8897.042} C_VEL
LIN {X 0,Y 450.226,Z 406.444,A -85,B 0,C 180,E1 -8897.579,E2 -8897.579} C_VEL
LIN {X 0,Y 450.006,Z 418.578,A -85,B 0,C 180,E1 -8898.12,E2 -8898.12} C_VEL
LIN {X 0,Y 449.625,Z 430.669,A -85,B 0,C 180,E1 -8898.848,E2 -8898.848} C_VEL
LIN {X 0,Y 449.161,Z 442.197,A -85,B 0,C 180,E1 -8899.749,E2 -8899.749} C_VEL
LIN {X 0,Y 448.824,Z 448.411,A -85,B 0,C 180,E1 -8900.337,E2 -8900.337} C_VEL
LIN {X 0,Y 447.987,Z 453.021,A -85,B 0,C 180,E1 -8900.797,E2 -8900.797} C_VEL
LIN {X 0,Y 444.855,Z 460.34,A -85,B 0,C 180,E1 -8901.555,E2 -8901.555} C_VEL
LIN {X 0,Y 441.681,Z 467.111,A -85,B 0,C 180,E1 -8902.394,E2 -8902.394} C_VEL
LIN {X 0,Y 440.79,Z 470.851,A -85,B 0,C 180,E1 -8902.974,E2 -8902.974} C_VEL
LIN {X 0,Y 440.241,Z 477.827,A -85,B 0,C 180,E1 -8904.275,E2 -8904.275} C_VEL
LIN {X 0,Y 439.9,Z 484.583,A -85,B 0,C 180,E1 -8905.878,E2 -8905.878} C_VEL
LIN {X 0,Y 439.589,Z 489.082,A -85,B 0,C 180,E1 -8907.252,E2 -8907.252} C_VEL
LIN {X 0,Y 439.434,Z 491.484,A -85,B 0,C 180,E1 -8908.168,E2 -8908.168} C_VEL
LIN {X 0,Y 439.212,Z 494.952,A -85,B 0,C 180,E1 -8910.001,E2 -8910.001} C_VEL
LIN {X 0,Y 439.07,Z 496.11,A -85,B 0,C 180,E1 -8910.918,E2 -8910.918} C_VEL
LIN {X 0,Y 439.137,Z 496.811,A -85,B 0,C 180,E1 -8911.835,E2 -8911.835} C_VEL
LIN {X 0,Y 439.072,Z 497.131,A -85,B 0,C 180,E1 -8913.672,E2 -8913.672} C_VEL
LIN {X 0,Y 439.143,Z 496.713,A -85,B 0,C 180,E1 -8914.591,E2 -8914.591} C_VEL
LIN {X 0,Y 439.305,Z 495.862,A -85,B 0,C 180,E1 -8915.509,E2 -8915.509} C_VEL
LIN {X 0,Y 439.421,Z 493.05,A -85,B 0,C 180,E1 -8917.352,E2 -8917.352} C_VEL
LIN {X 0,Y 439.643,Z 489.793,A -85,B 0,C 180,E1 -8918.736,E2 -8918.736} C_VEL
LIN {X 0,Y 440.023,Z 485.463,A -85,B 0,C 180,E1 -8920.12,E2 -8920.12} C_VEL
LIN {X 0,Y 440.418,Z 478.866,A -85,B 0,C 180,E1 -8921.74,E2 -8921.74} C_VEL
LIN {X 0,Y 440.818,Z 471.887,A -85,B 0,C 180,E1 -8923.096,E2 -8923.096} C_VEL
LIN {X 0,Y 441.416,Z 464.298,A -85,B 0,C 180,E1 -8924.288,E2 -8924.288} C_VEL
LIN {X 0,Y 441.991,Z 454.272,A -85,B 0,C 180,E1 -8925.565,E2 -8925.565} C_VEL
LIN {X 0,Y 442.516,Z 444.059,A -85,B 0,C 180,E1 -8926.612,E2 -8926.612} C_VEL
LIN {X 0,Y 443.051,Z 432.591,A -85,B 0,C 180,E1 -8927.542,E2 -8927.542} C_VEL
LIN {X 0,Y 443.522,Z 421.027,A -85,B 0,C 180,E1 -8928.263,E2 -8928.263} C_VEL
LIN {X 0,Y 443.714,Z 408.137,A -85,B 0,C 180,E1 -8928.868,E2 -8928.868} C_VEL
LIN {X 0,Y 439.576,Z 395.951,A -85,B 0,C 180,E1 -8929.433,E2 -8929.433} C_VEL
LIN {X 0,Y 439.189,Z 394.406,A -85,B 0,C 180,E1 -8929.505,E2 -8929.505} C_VEL
LIN {X 0,Y 439.355,Z 394.381,A -85,B 0,C 180,E1 -8931.908,E2 -8931.908} C_VEL
LIN {X 0,Y 439.422,Z 394.373,A -85,B 0,C 180,E1 -8934.573,E2 -8934.573} C_VEL
LIN {X 0,Y 439.448,Z 394.369,A -85,B 0,C 180,E1 -8937.633,E2 -8937.633} C_VEL
LIN {X 0,Y 439.367,Z 394.384,A -85,B 0,C 180,E1 -8940.789,E2 -8940.789} C_VEL
LIN {X 0,Y 439.39,Z 394.378,A -85,B 0,C 180,E1 -8944.044,E2 -8944.044} C_VEL
LIN {X 0,Y 439.354,Z 394.379,A -85,B 0,C 180,E1 -8946.887,E2 -8946.887} C_VEL
LIN {X 0,Y 439.407,Z 394.371,A -85,B 0,C 180,E1 -8949.849,E2 -8949.849} C_VEL
LIN {X 0,Y 439.387,Z 394.378,A -85,B 0,C 180,E1 -8952.627,E2 -8952.627} C_VEL
LIN {X 0,Y 439.411,Z 394.37,A -85,B 0,C 180,E1 -8955.271,E2 -8955.271} C_VEL
LIN {X 0,Y 439.395,Z 394.372,A -85,B 0,C 180,E1 -8958.743,E2 -8958.743} C_VEL
LIN {X 0,Y 439.387,Z 394.357,A -85,B 0,C 180,E1 -8961.606,E2 -8961.606} C_VEL
LIN {X 0,Y 439.406,Z 394.373,A -85,B 0,C 180,E1 -8964.844,E2 -8964.844} C_VEL
LIN {X 0,Y 439.377,Z 394.368,A -85,B 0,C 180,E1 -8968.139,E2 -8968.139} C_VEL
LIN {X 0,Y 439.437,Z 394.35,A -85,B 0,C 180,E1 -8971.598,E2 -8971.598} C_VEL
LIN {X 0,Y 439.402,Z 394.373,A -85,B 0,C 180,E1 -8974.415,E2 -8974.415} C_VEL
LIN {X 0,Y 439.368,Z 394.383,A -85,B 0,C 180,E1 -8977.424,E2 -8977.424} C_VEL
LIN {X 0,Y 439.445,Z 394.369,A -85,B 0,C 180,E1 -8980.663,E2 -8980.663} C_VEL
LIN {X 0,Y 439.406,Z 394.375,A -85,B 0,C 180,E1 -8982.42,E2 -8982.42} C_VEL
LIN {X 0,Y 443.886,Z 408.964,A -85,B 0,C 180,E1 -8983.441,E2 -8983.441} C_VEL
LIN {X 0,Y 443.576,Z 420.637,A -85,B 0,C 180,E1 -8984.256,E2 -8984.256} C_VEL
LIN {X 0,Y 442.881,Z 432.925,A -85,B 0,C 180,E1 -8985.291,E2 -8985.291} C_VEL
LIN {X 0,Y 442.19,Z 444.126,A -85,B 0,C 180,E1 -8986.442,E2 -8986.442} C_VEL
LIN {X 0,Y 441.392,Z 455.154,A -85,B 0,C 180,E1 -8987.82,E2 -8987.82} C_VEL
LIN {X 0,Y 440.806,Z 464.277,A -85,B 0,C 180,E1 -8989.202,E2 -8989.202} C_VEL
LIN {X 0,Y 440.295,Z 473.016,A -85,B 0,C 180,E1 -8990.815,E2 -8990.815} C_VEL
LIN {X 0,Y 439.844,Z 480.384,A -85,B 0,C 180,E1 -8992.497,E2 -8992.497} C_VEL
LIN {X 0,Y 439.543,Z 485.741,A -85,B 0,C 180,E1 -8994.034,E2 -8994.034} C_VEL
LIN {X 0,Y 439.359,Z 490.668,A -85,B 0,C 180,E1 -8995.872,E2 -8995.872} C_VEL
LIN {X 0,Y 439.087,Z 493.357,A -85,B 0,C 180,E1 -8997.247,E2 -8997.247} C_VEL
LIN {X 0,Y 439.043,Z 495.748,A -85,B 0,C 180,E1 -8999.083,E2 -8999.083} C_VEL
LIN {X 0,Y 439.091,Z 496.797,A -85,B 0,C 180,E1 -9000.917,E2 -9000.917} C_VEL
LIN {X 0,Y 439.212,Z 496.517,A -85,B 0,C 180,E1 -9002.751,E2 -9002.751} C_VEL
LIN {X 0,Y 439.291,Z 494.902,A -85,B 0,C 180,E1 -9004.588,E2 -9004.588} C_VEL
LIN {X 0,Y 439.651,Z 491.878,A -85,B 0,C 180,E1 -9006.425,E2 -9006.425} C_VEL
LIN {X 0,Y 439.971,Z 487.409,A -85,B 0,C 180,E1 -9008.266,E2 -9008.266} C_VEL
LIN {X 0,Y 440.407,Z 481.335,A -85,B 0,C 180,E1 -9010.11,E2 -9010.11} C_VEL
LIN {X 0,Y 440.949,Z 474.477,A -85,B 0,C 180,E1 -9011.725,E2 -9011.725} C_VEL
LIN {X 0,Y 441.718,Z 465.835,A -85,B 0,C 180,E1 -9013.338,E2 -9013.338} C_VEL
LIN {X 0,Y 442.448,Z 456.79,A -85,B 0,C 180,E1 -9014.723,E2 -9014.723} C_VEL
LIN {X 0,Y 443.175,Z 446.803,A -85,B 0,C 180,E1 -9015.994,E2 -9015.994} C_VEL
LIN {X 0,Y 443.935,Z 435.797,A -85,B 0,C 180,E1 -9017.149,E2 -9017.149} C_VEL
LIN {X 0,Y 444.716,Z 423.703,A -85,B 0,C 180,E1 -9018.184,E2 -9018.184} C_VEL
LIN {X 0,Y 445.359,Z 412.436,A -85,B 0,C 180,E1 -9018.962,E2 -9018.962} C_VEL
LIN {X 0,Y 444.685,Z 409.15,A -85,B 0,C 180,E1 -9019.21,E2 -9019.21} C_VEL
LIN {X 0,Y 441.234,Z 399.281,A -85,B 0,C 180,E1 -9019.989,E2 -9019.989} C_VEL
LIN {X 0,Y 439.407,Z 394.382,A -85,B 0,C 180,E1 -9020.358,E2 -9020.358} C_VEL
LIN {X 0,Y 439.39,Z 394.382,A -85,B 0,C 180,E1 -9023.57,E2 -9023.57} C_VEL
LIN {X 0,Y 439.432,Z 394.376,A -85,B 0,C 180,E1 -9026.603,E2 -9026.603} C_VEL
LIN {X 0,Y 439.385,Z 394.38,A -85,B 0,C 180,E1 -9029.726,E2 -9029.726} C_VEL
LIN {X 0,Y 439.376,Z 394.382,A -85,B 0,C 180,E1 -9032.946,E2 -9032.946} C_VEL
LIN {X 0,Y 439.376,Z 394.381,A -85,B 0,C 180,E1 -9036.287,E2 -9036.287} C_VEL
LIN {X 0,Y 439.409,Z 394.378,A -85,B 0,C 180,E1 -9039.849,E2 -9039.849} C_VEL
LIN {X 0,Y 439.385,Z 394.381,A -85,B 0,C 180,E1 -9042.627,E2 -9042.627} C_VEL
LIN {X 0,Y 439.422,Z 394.524,A -85,B 0,C 180,E1 -9045.715,E2 -9045.715} C_VEL
LIN {X 0,Y 440.782,Z 401.046,A -85,B 0,C 180,E1 -9048.537,E2 -9048.537} C_VEL
LIN {X 0,Y 441.735,Z 406.282,A -85,B 0,C 180,E1 -9050.475,E2 -9050.475} C_VEL
LIN {X 0,Y 441.707,Z 409.88,A -85,B 0,C 180,E1 -9051.645,E2 -9051.645} C_VEL
LIN {X 0,Y 440.546,Z 423.186,A -85,B 0,C 180,E1 -9055.505,E2 -9055.505} C_VEL
LIN {X 0,Y 440.145,Z 435.299,A -85,B 0,C 180,E1 -9058.738,E2 -9058.738} C_VEL
LIN {X 0,Y 439.858,Z 446.229,A -85,B 0,C 180,E1 -9061.496,E2 -9061.496} C_VEL
LIN {X 0,Y 439.594,Z 460.384,A -85,B 0,C 180,E1 -9064.933,E2 -9064.933} C_VEL
LIN {X 0,Y 439.336,Z 473.8,A -85,B 0,C 180,E1 -9068.097,E2 -9068.097} C_VEL
LIN {X 0,Y 439.264,Z 481.871,A -85,B 0,C 180,E1 -9069.925,E2 -9069.925} C_VEL
LIN {X 0,Y 441.414,Z 498.269,A -85,B 0,C 180,E1 -9070.5,E2 -9070.5} C_VEL
LIN {X 0,Y 442.413,Z 514.163,A -85,B 0,C 180,E1 -9071.196,E2 -9071.196} C_VEL
LIN {X 0,Y 443.311,Z 523.166,A -85,B 0,C 180,E1 -9071.693,E2 -9071.693} C_VEL
LIN {X 0,Y 442.44,Z 537.539,A -85,B 0,C 180,E1 -9072.552,E2 -9072.552} C_VEL
LIN {X 0,Y 441.623,Z 549.923,A -85,B 0,C 180,E1 -9073.472,E2 -9073.472} C_VEL
LIN {X 0,Y 440.786,Z 562.723,A -85,B 0,C 180,E1 -9074.628,E2 -9074.628} C_VEL
LIN {X 0,Y 440.073,Z 574.373,A -85,B 0,C 180,E1 -9075.903,E2 -9075.903} C_VEL
LIN {X 0,Y 439.591,Z 584.464,A -85,B 0,C 180,E1 -9077.224,E2 -9077.224} C_VEL
LIN {X 0,Y 439.225,Z 593.873,A -85,B 0,C 180,E1 -9078.695,E2 -9078.695} C_VEL
LIN {X 0,Y 438.945,Z 602.438,A -85,B 0,C 180,E1 -9080.321,E2 -9080.321} C_VEL
LIN {X 0,Y 438.832,Z 608.474,A -85,B 0,C 180,E1 -9081.712,E2 -9081.712} C_VEL
LIN {X 0,Y 438.798,Z 614.862,A -85,B 0,C 180,E1 -9083.562,E2 -9083.562} C_VEL
LIN {X 0,Y 438.889,Z 619.567,A -85,B 0,C 180,E1 -9085.407,E2 -9085.407} C_VEL
LIN {X 0,Y 438.804,Z 622.676,A -85,B 0,C 180,E1 -9087.245,E2 -9087.245} C_VEL
LIN {X 0,Y 438.798,Z 624.298,A -85,B 0,C 180,E1 -9089.081,E2 -9089.081} C_VEL
LIN {X 0,Y 438.916,Z 624.575,A -85,B 0,C 180,E1 -9089.999,E2 -9089.999} C_VEL
LIN {X 0,Y 438.75,Z 623.981,A -85,B 0,C 180,E1 -9091.835,E2 -9091.835} C_VEL
LIN {X 0,Y 438.756,Z 621.96,A -85,B 0,C 180,E1 -9093.673,E2 -9093.673} C_VEL
LIN {X 0,Y 438.69,Z 618.434,A -85,B 0,C 180,E1 -9095.515,E2 -9095.515} C_VEL
LIN {X 0,Y 438.698,Z 614.783,A -85,B 0,C 180,E1 -9096.899,E2 -9096.899} C_VEL
LIN {X 0,Y 438.723,Z 610.129,A -85,B 0,C 180,E1 -9098.288,E2 -9098.288} C_VEL
LIN {X 0,Y 438.876,Z 603.385,A -85,B 0,C 180,E1 -9099.912,E2 -9099.912} C_VEL
LIN {X 0,Y 439.232,Z 594.996,A -85,B 0,C 180,E1 -9101.536,E2 -9101.536} C_VEL
LIN {X 0,Y 439.666,Z 586.237,A -85,B 0,C 180,E1 -9102.93,E2 -9102.93} C_VEL
LIN {X 0,Y 440.289,Z 575.665,A -85,B 0,C 180,E1 -9104.323,E2 -9104.323} C_VEL
LIN {X 0,Y 441.01,Z 563.9,A -85,B 0,C 180,E1 -9105.599,E2 -9105.599} C_VEL
LIN {X 0,Y 441.889,Z 552.251,A -85,B 0,C 180,E1 -9106.634,E2 -9106.634} C_VEL
LIN {X 0,Y 442.719,Z 539.578,A -85,B 0,C 180,E1 -9107.554,E2 -9107.554} C_VEL
LIN {X 0,Y 443.508,Z 525.304,A -85,B 0,C 180,E1 -9108.37,E2 -9108.37} C_VEL
LIN {X 0,Y 443.449,Z 521.153,A -85,B 0,C 180,E1 -9108.571,E2 -9108.571} C_VEL
LIN {X 0,Y 441.78,Z 506.295,A -85,B 0,C 180,E1 -9109.227,E2 -9109.227} C_VEL
LIN {X 0,Y 439.45,Z 490.427,A -85,B 0,C 180,E1 -9109.739,E2 -9109.739} C_VEL
LIN {X 0,Y 439.417,Z 489.485,A -85,B 0,C 180,E1 -9109.783,E2 -9109.783} C_VEL
LIN {X 0,Y 439.866,Z 476.526,A -85,B 0,C 180,E1 -9113.043,E2 -9113.043} C_VEL
LIN {X 0,Y 440.475,Z 462.312,A -85,B 0,C 180,E1 -9116.683,E2 -9116.683} C_VEL
LIN {X 0,Y 441.319,Z 447.015,A -85,B 0,C 180,E1 -9120.689,E2 -9120.689} C_VEL
LIN {X 0,Y 442.132,Z 432.82,A -85,B 0,C 180,E1 -9124.522,E2 -9124.522} C_VEL
LIN {X 0,Y 443.233,Z 418.116,A -85,B 0,C 180,E1 -9128.619,E2 -9128.619} C_VEL
LIN {X 0,Y 443.312,Z 413.831,A -85,B 0,C 180,E1 -9129.864,E2 -9129.864} C_VEL
LIN {X 0,Y 441.799,Z 405.722,A -85,B 0,C 180,E1 -9132.4,E2 -9132.4} C_VEL
LIN {X 0,Y 439.406,Z 394.377,A -85,B 0,C 180,E1 -9136.152,E2 -9136.152} C_VEL
LIN {X 0,Y 439.393,Z 394.378,A -85,B 0,C 180,E1 -9139.021,E2 -9139.021} C_VEL
LIN {X 0,Y 439.386,Z 394.381,A -85,B 0,C 180,E1 -9141.603,E2 -9141.603} C_VEL
LIN {X 0,Y 439.392,Z 394.377,A -85,B 0,C 180,E1 -9144.843,E2 -9144.843} C_VEL
LIN {X 0,Y 439.365,Z 394.379,A -85,B 0,C 180,E1 -9148.139,E2 -9148.139} C_VEL
LIN {X 0,Y 439.415,Z 394.377,A -85,B 0,C 180,E1 -9151.327,E2 -9151.327} C_VEL
LIN {X 0,Y 439.395,Z 394.376,A -85,B 0,C 180,E1 -9154.415,E2 -9154.415} C_VEL
LIN {X 0,Y 439.354,Z 394.384,A -85,B 0,C 180,E1 -9157.424,E2 -9157.424} C_VEL
LIN {X 0,Y 439.431,Z 394.372,A -85,B 0,C 180,E1 -9160.662,E2 -9160.662} C_VEL
LIN {X 0,Y 439.452,Z 394.369,A -85,B 0,C 180,E1 -9164.224,E2 -9164.224} C_VEL
LIN {X 0,Y 439.497,Z 394.363,A -85,B 0,C 180,E1 -9168.002,E2 -9168.002} C_VEL
LIN {X 0,Y 439.537,Z 394.358,A -85,B 0,C 180,E1 -9171.726,E2 -9171.726} C_VEL
LIN {X 0,Y 439.611,Z 394.349,A -85,B 0,C 180,E1 -9174.496,E2 -9174.496} C_VEL
LIN {X 0,Y 439.626,Z 394.347,A -85,B 0,C 180,E1 -9178.168,E2 -9178.168} C_VEL
LIN {X 0,Y 439.754,Z 394.331,A -85,B 0,C 180,E1 -9180,E2 -9180} C_VEL
LIN {X 0,Y 439.647,Z 394.346,A -85,B 0,C 180,E1 -9182.749,E2 -9182.749} C_VEL
LIN {X 0,Y 439.61,Z 394.35,A -85,B 0,C 180,E1 -9186.426,E2 -9186.426} C_VEL
LIN {X 0,Y 439.492,Z 394.366,A -85,B 0,C 180,E1 -9189.202,E2 -9189.202} C_VEL
LIN {X 0,Y 439.494,Z 394.365,A -85,B 0,C 180,E1 -9192.727,E2 -9192.727} C_VEL
LIN {X 0,Y 439.437,Z 394.371,A -85,B 0,C 180,E1 -9196.35,E2 -9196.35} C_VEL
LIN {X 0,Y 439.393,Z 394.376,A -85,B 0,C 180,E1 -9199.627,E2 -9199.627} C_VEL
LIN {X 0,Y 439.356,Z 394.382,A -85,B 0,C 180,E1 -9202.576,E2 -9202.576} C_VEL
LIN {X 0,Y 439.397,Z 394.375,A -85,B 0,C 180,E1 -9205.586,E2 -9205.586} C_VEL
LIN {X 0,Y 439.409,Z 394.376,A -85,B 0,C 180,E1 -9208.674,E2 -9208.674} C_VEL
LIN {X 0,Y 439.363,Z 394.381,A -85,B 0,C 180,E1 -9212.032,E2 -9212.032} C_VEL
LIN {X 0,Y 439.389,Z 394.377,A -85,B 0,C 180,E1 -9215.342,E2 -9215.342} C_VEL
LIN {X 0,Y 439.384,Z 394.379,A -85,B 0,C 180,E1 -9218.595,E2 -9218.595} C_VEL
LIN {X 0,Y 439.384,Z 394.378,A -85,B 0,C 180,E1 -9221.258,E2 -9221.258} C_VEL
LIN {X 0,Y 439.401,Z 394.379,A -85,B 0,C 180,E1 -9224.73,E2 -9224.73} C_VEL
LIN {X 0,Y 439.393,Z 394.376,A -85,B 0,C 180,E1 -9227.797,E2 -9227.797} C_VEL
LIN {X 0,Y 439.448,Z 394.37,A -85,B 0,C 180,E1 -9230.232,E2 -9230.232} C_VEL
LIN {X 0,Y 439.375,Z 394.379,A -85,B 0,C 180,E1 -9233.715,E2 -9233.715} C_VEL
LIN {X 0,Y 439.37,Z 394.38,A -85,B 0,C 180,E1 -9237.055,E2 -9237.055} C_VEL
LIN {X 0,Y 439.382,Z 394.379,A -85,B 0,C 180,E1 -9240.276,E2 -9240.276} C_VEL
LIN {X 0,Y 439.429,Z 394.371,A -85,B 0,C 180,E1 -9243.398,E2 -9243.398} C_VEL
LIN {X 0,Y 439.387,Z 394.379,A -85,B 0,C 180,E1 -9246.431,E2 -9246.431} C_VEL
LIN {X 0,Y 439.389,Z 394.376,A -85,B 0,C 180,E1 -9249.398,E2 -9249.398} C_VEL
LIN {X 0,Y 439.429,Z 394.373,A -85,B 0,C 180,E1 -9252.311,E2 -9252.311} C_VEL
LIN {X 0,Y 439.354,Z 394.383,A -85,B 0,C 180,E1 -9255.172,E2 -9255.172} C_VEL
LIN {X 0,Y 439.264,Z 394.397,A -85,B 0,C 180,E1 -9256.798,E2 -9256.798} C_VEL
LIN {X 0,Y 443.303,Z 407.482,A -85,B 0,C 180,E1 -9257.35,E2 -9257.35} C_VEL
LIN {X 0,Y 443.222,Z 418.779,A -85,B 0,C 180,E1 -9257.859,E2 -9257.859} C_VEL
LIN {X 0,Y 442.842,Z 430.472,A -85,B 0,C 180,E1 -9258.559,E2 -9258.559} C_VEL
LIN {X 0,Y 442.345,Z 442.278,A -85,B 0,C 180,E1 -9259.473,E2 -9259.473} C_VEL
LIN {X 0,Y 441.746,Z 453.07,A -85,B 0,C 180,E1 -9260.541,E2 -9260.541} C_VEL
LIN {X 0,Y 441.181,Z 462.921,A -85,B 0,C 180,E1 -9261.758,E2 -9261.758} C_VEL
LIN {X 0,Y 440.79,Z 470.851,A -85,B 0,C 180,E1 -9262.974,E2 -9262.974} C_VEL
LIN {X 0,Y 439.906,Z 474.439,A -85,B 0,C 180,E1 -9263.578,E2 -9263.578} C_VEL
LIN {X 0,Y 436.74,Z 479.973,A -85,B 0,C 180,E1 -9264.568,E2 -9264.568} C_VEL
LIN {X 0,Y 433.584,Z 484.908,A -85,B 0,C 180,E1 -9265.62,E2 -9265.62} C_VEL
LIN {X 0,Y 432.731,Z 487.452,A -85,B 0,C 180,E1 -9266.316,E2 -9266.316} C_VEL
LIN {X 0,Y 432.546,Z 491.406,A -85,B 0,C 180,E1 -9267.673,E2 -9267.673} C_VEL
LIN {X 0,Y 432.285,Z 494.482,A -85,B 0,C 180,E1 -9269.069,E2 -9269.069} C_VEL
LIN {X 0,Y 432.197,Z 496.005,A -85,B 0,C 180,E1 -9270.001,E2 -9270.001} C_VEL
LIN {X 0,Y 432.048,Z 497.146,A -85,B 0,C 180,E1 -9270.933,E2 -9270.933} C_VEL
LIN {X 0,Y 432.116,Z 497.831,A -85,B 0,C 180,E1 -9271.865,E2 -9271.865} C_VEL
LIN {X 0,Y 432.048,Z 498.13,A -85,B 0,C 180,E1 -9273.732,E2 -9273.732} C_VEL
LIN {X 0,Y 432.127,Z 497.691,A -85,B 0,C 180,E1 -9274.665,E2 -9274.665} C_VEL
LIN {X 0,Y 432.302,Z 496.827,A -85,B 0,C 180,E1 -9275.599,E2 -9275.599} C_VEL
LIN {X 0,Y 432.431,Z 493.99,A -85,B 0,C 180,E1 -9277.472,E2 -9277.472} C_VEL
LIN {X 0,Y 432.688,Z 490.708,A -85,B 0,C 180,E1 -9278.877,E2 -9278.877} C_VEL
LIN {X 0,Y 433.093,Z 486.347,A -85,B 0,C 180,E1 -9280.283,E2 -9280.283} C_VEL
LIN {X 0,Y 433.513,Z 479.712,A -85,B 0,C 180,E1 -9281.93,E2 -9281.93} C_VEL
LIN {X 0,Y 433.933,Z 472.767,A -85,B 0,C 180,E1 -9283.295,E2 -9283.295} C_VEL
LIN {X 0,Y 434.569,Z 465.071,A -85,B 0,C 180,E1 -9284.518,E2 -9284.518} C_VEL
LIN {X 0,Y 435.197,Z 454.972,A -85,B 0,C 180,E1 -9285.815,E2 -9285.815} C_VEL
LIN {X 0,Y 435.749,Z 444.696,A -85,B 0,C 180,E1 -9286.878,E2 -9286.878} C_VEL
LIN {X 0,Y 436.272,Z 434.75,A -85,B 0,C 180,E1 -9287.703,E2 -9287.703} C_VEL
LIN {X 0,Y 436.733,Z 423.512,A -85,B 0,C 180,E1 -9288.437,E2 -9288.437} C_VEL
LIN {X 0,Y 437.016,Z 410.437,A -85,B 0,C 180,E1 -9289.077,E2 -9289.077} C_VEL
LIN {X 0,Y 434.301,Z 401.623,A -85,B 0,C 180,E1 -9289.516,E2 -9289.516} C_VEL
LIN {X 0,Y 432.197,Z 395.277,A -85,B 0,C 180,E1 -9289.797,E2 -9289.797} C_VEL
LIN {X 0,Y 432.315,Z 395.26,A -85,B 0,C 180,E1 -9292.965,E2 -9292.965} C_VEL
LIN {X 0,Y 432.358,Z 395.252,A -85,B 0,C 180,E1 -9295.002,E2 -9295.002} C_VEL
LIN {X 0,Y 432.388,Z 395.248,A -85,B 0,C 180,E1 -9298.124,E2 -9298.124} C_VEL
LIN {X 0,Y 432.327,Z 395.259,A -85,B 0,C 180,E1 -9301.346,E2 -9301.346} C_VEL
LIN {X 0,Y 432.343,Z 395.258,A -85,B 0,C 180,E1 -9304.678,E2 -9304.678} C_VEL
LIN {X 0,Y 432.342,Z 395.248,A -85,B 0,C 180,E1 -9308.15,E2 -9308.15} C_VEL
LIN {X 0,Y 432.338,Z 395.253,A -85,B 0,C 180,E1 -9311.602,E2 -9311.602} C_VEL
LIN {X 0,Y 432.339,Z 395.259,A -85,B 0,C 180,E1 -9314.347,E2 -9314.347} C_VEL
LIN {X 0,Y 432.33,Z 395.255,A -85,B 0,C 180,E1 -9317.015,E2 -9317.015} C_VEL
LIN {X 0,Y 432.339,Z 395.248,A -85,B 0,C 180,E1 -9319.821,E2 -9319.821} C_VEL
LIN {X 0,Y 432.321,Z 395.249,A -85,B 0,C 180,E1 -9323.023,E2 -9323.023} C_VEL
LIN {X 0,Y 432.365,Z 395.255,A -85,B 0,C 180,E1 -9325.996,E2 -9325.996} C_VEL
LIN {X 0,Y 432.352,Z 395.234,A -85,B 0,C 180,E1 -9329.49,E2 -9329.49} C_VEL
LIN {X 0,Y 432.395,Z 395.238,A -85,B 0,C 180,E1 -9332.928,E2 -9332.928} C_VEL
LIN {X 0,Y 432.372,Z 395.253,A -85,B 0,C 180,E1 -9336.023,E2 -9336.023} C_VEL
LIN {X 0,Y 432.354,Z 395.253,A -85,B 0,C 180,E1 -9339.046,E2 -9339.046} C_VEL
LIN {X 0,Y 432.402,Z 395.41,A -85,B 0,C 180,E1 -9342.179,E2 -9342.179} C_VEL
LIN {X 0,Y 436.281,Z 408.005,A -85,B 0,C 180,E1 -9343.051,E2 -9343.051} C_VEL
LIN {X 0,Y 437.178,Z 411.304,A -85,B 0,C 180,E1 -9343.3,E2 -9343.3} C_VEL
LIN {X 0,Y 436.61,Z 424.155,A -85,B 0,C 180,E1 -9344.238,E2 -9344.238} C_VEL
LIN {X 0,Y 435.821,Z 436.711,A -85,B 0,C 180,E1 -9345.366,E2 -9345.366} C_VEL
LIN {X 0,Y 435.208,Z 446.76,A -85,B 0,C 180,E1 -9346.458,E2 -9346.458} C_VEL
LIN {X 0,Y 434.388,Z 457.526,A -85,B 0,C 180,E1 -9347.858,E2 -9347.858} C_VEL
LIN {X 0,Y 433.837,Z 466.428,A -85,B 0,C 180,E1 -9349.263,E2 -9349.263} C_VEL
LIN {X 0,Y 433.277,Z 474.989,A -85,B 0,C 180,E1 -9350.9,E2 -9350.9} C_VEL
LIN {X 0,Y 432.854,Z 481.897,A -85,B 0,C 180,E1 -9352.536,E2 -9352.536} C_VEL
LIN {X 0,Y 432.556,Z 486.662,A -85,B 0,C 180,E1 -9353.937,E2 -9353.937} C_VEL
LIN {X 0,Y 432.358,Z 491.63,A -85,B 0,C 180,E1 -9355.805,E2 -9355.805} C_VEL
LIN {X 0,Y 432.067,Z 494.356,A -85,B 0,C 180,E1 -9357.203,E2 -9357.203} C_VEL
LIN {X 0,Y 432.024,Z 496.776,A -85,B 0,C 180,E1 -9359.068,E2 -9359.068} C_VEL
LIN {X 0,Y 432.093,Z 497.855,A -85,B 0,C 180,E1 -9360.932,E2 -9360.932} C_VEL
LIN {X 0,Y 432.21,Z 497.615,A -85,B 0,C 180,E1 -9362.796,E2 -9362.796} C_VEL
LIN {X 0,Y 432.301,Z 496.042,A -85,B 0,C 180,E1 -9364.662,E2 -9364.662} C_VEL
LIN {X 0,Y 432.681,Z 493.043,A -85,B 0,C 180,E1 -9366.528,E2 -9366.528} C_VEL
LIN {X 0,Y 433.052,Z 488.591,A -85,B 0,C 180,E1 -9368.399,E2 -9368.399} C_VEL
LIN {X 0,Y 433.53,Z 482.534,A -85,B 0,C 180,E1 -9370.272,E2 -9370.272} C_VEL
LIN {X 0,Y 434.105,Z 475.714,A -85,B 0,C 180,E1 -9371.912,E2 -9371.912} C_VEL
LIN {X 0,Y 434.933,Z 467.15,A -85,B 0,C 180,E1 -9373.55,E2 -9373.55} C_VEL
LIN {X 0,Y 435.721,Z 458.165,A -85,B 0,C 180,E1 -9374.956,E2 -9374.956} C_VEL
LIN {X 0,Y 436.568,Z 447.218,A -85,B 0,C 180,E1 -9376.363,E2 -9376.363} C_VEL
LIN {X 0,Y 437.405,Z 436.052,A -85,B 0,C 180,E1 -9377.533,E2 -9377.533} C_VEL
LIN {X 0,Y 438.235,Z 423.534,A -85,B 0,C 180,E1 -9378.607,E2 -9378.607} C_VEL
LIN {X 0,Y 438.764,Z 413.106,A -85,B 0,C 180,E1 -9379.341,E2 -9379.341} C_VEL
LIN {X 0,Y 435.357,Z 402.999,A -85,B 0,C 180,E1 -9380.175,E2 -9380.175} C_VEL
